EMstopSwitch(			TriggerInput := NOT (get.b_EstopChannelAOK AND get.b_EstopChannelBOK), 
						LogItemGroup :=  eLogItemGroupID.Safety, 
						LogItemName := 'EmStopSwCnt', 
						LogType := eLogTypes.TrackCycles);

SafetyStopCount(		TriggerInput := get.b_SafetyOK, 
						LogItemGroup :=  eLogItemGroupID.Safety, 
						LogItemName := 'SafetyStopCnt', 
						LogType := eLogTypes.TrackCycles);
END_METHOD

METHOD Reset : BOOL
VAR_INPUT
	prgReset: BOOL;
END_VAR
IF ton_Reset.Q THEN
	ToSafetyPrg.b_safetyPRGReset := FALSE;
	ToSafetyPrg.b_ErrorReset := FALSE;
	ton_Reset.IN := FALSE;
	Reset := get.b_SafetyOK;
ELSE
	ton_Reset.IN :=TRUE;
	ToSafetyPrg.b_safetyPRGReset := prgReset;
	ToSafetyPrg.b_ErrorReset := TRUE;
END_IF
END_METHOD

END_PROGRAM

// ---- POUs/Objects/WearLogging/FB_Varlogger.TcPOU
//FB for complex logvalues
//Can keep track of on-time, rising edge count, highest/lowest value and actual values
//Simple overwriting and min/max of variables can also be done without this by calling the Wearlogging methods directly

FUNCTION_BLOCK FB_Varlogger
VAR_INPUT
	LogItemGroup	:	eLogItemGroupID;		//Json itemgroup
	LogItemName		:	STRING;					//Json itemname
	LogType			:	eLogTypes;				//Determines logging functionality
	
	TriggerInput	:	BOOL;					//boolean input for trackcycles and trackOnTime
	NewValue		:	ANY;					//New value for 
END_VAR

VAR
	rtrig_InputValue		:	r_trig;
	ton_IncrementingTimer	:	ton	:=	(pt := T#15M);
	ftrig_timerloss			:	f_trig;
	rtrig_TimerDone			:	r_trig;
	elapsedTime				:	TIME;	
	
	ton_UpdateTimer			:	Ton;
	LrealPointer			: 	POINTER TO LREAL;
	realPointer				:	POINTER TO REAL;
	StringPointer			:	POINTER TO STRING;
	
	USINTPOINTER			: 	POINTER TO USINT;
	UINTPOINTER				: 	POINTER TO UINT;
	UDINTPOINTER			: 	POINTER TO UDINT;
	ULINTPOINTER			: 	POINTER TO ULINT;
	SINTPOINTER				: 	POINTER TO SINT;
	INTPOINTER				: 	POINTER TO INT;
	DINTPOINTER				: 	POINTER TO DINT;
	LINTPOINTER				: 	POINTER TO LINT;	

	TempString				:	String;	
END_VAR

CASE LogType OF 
	eLogTypes.TrackCycles:
		rtrig_InputValue(clk := TriggerInput);
		IF rtrig_InputValue.Q AND NOT gvl.b_Initcycle THEN
			WearLogging.SetInteger(LogItemGroup, LogItemName, LogType, 1);
		END_IF

	eLogTypes.TrackOnTime:
		ton_IncrementingTimer	(in := TriggerInput AND NOT ton_incrementingTimer.Q);
		ftrig_timerloss(clk := TriggerInput);
		rtrig_timerDone(clk := ton_IncrementingTimer.Q);
		
		IF ftrig_timerloss.Q THEN
			WearLogging.setFloat(LogItemGroup, LogItemName, LogType, TO_LREAL(TIME_TO_LREAL(elapsedTime)/TIME_TO_LREAL(T#1H)));
		END_IF
		
		IF rtrig_timerDone.Q THEN
			elapsedTime := ton_IncrementingTimer.PT;
			WearLogging.setFloat(LogItemGroup, LogItemName, LogType, TO_LREAL(TIME_TO_LREAL(elapsedTime)/TIME_TO_LREAL(T#1H)));
		END_IF
		
		elapsedTime := ton_IncrementingTimer.ET;
		
	eLogTypes.WriteValue, eLogTypes.KeepHighestValue, eLogTypes.KeepLowestValue:
		IF TriggerInput and not gvl.b_initCycle then	
		
			CASE NewValue.TypeClass OF
				__SYSTEM.TYPE_CLASS.TYPE_REAL:
					realPointer := NewValue.pValue;
					WearLogging.setFloat(LogItemGroup, LogItemName, LogType,TO_LREAL(realPointer^));
					
				__SYSTEM.TYPE_CLASS.TYPE_LREAL:
					LrealPointer := NewValue.pValue;
					WearLogging.setFloat(LogItemGroup, LogItemName, LogType,LrealPointer^);
					
				__SYSTEM.TYPE_CLASS.TYPE_USINT:
					USINTPOINTER := NewValue.pValue;
					WearLogging.setInteger(LogItemGroup, LogItemName, LogType, TO_LINT(USINTPOINTER^));
				
				__SYSTEM.TYPE_CLASS.TYPE_UINT:
					UINTPOINTER := NewValue.pValue;
					WearLogging.setInteger(LogItemGroup, LogItemName, LogType, TO_LINT(UINTPOINTER^));
				
				__SYSTEM.TYPE_CLASS.TYPE_UDINT:
					UDINTPOINTER := NewValue.pValue;
					WearLogging.setInteger(LogItemGroup, LogItemName, LogType, TO_LINT(UDINTPOINTER^));
				
				__SYSTEM.TYPE_CLASS.TYPE_ULINT:
					ULINTPOINTER := NewValue.pValue;
					WearLogging.setInteger(LogItemGroup, LogItemName, LogType, TO_LINT(ULINTPOINTER^));
				
				__SYSTEM.TYPE_CLASS.TYPE_SINT:
					SINTPOINTER := NewValue.pValue;
					WearLogging.setInteger(LogItemGroup, LogItemName, LogType, TO_LINT(SINTPOINTER^));
				
				__SYSTEM.TYPE_CLASS.TYPE_INT:
					INTPOINTER := NewValue.pValue;
					WearLogging.setInteger(LogItemGroup, LogItemName, LogType, TO_LINT(INTPOINTER^));
				
				__SYSTEM.TYPE_CLASS.TYPE_DINT:
					DINTPOINTER := NewValue.pValue;
					WearLogging.setInteger(LogItemGroup, LogItemName, LogType, TO_LINT(DINTPOINTER^));
				
				__SYSTEM.TYPE_CLASS.TYPE_LINT:
					LINTPOINTER := NewValue.pValue;
					WearLogging.setInteger(LogItemGroup, LogItemName, LogType, TO_LINT(LINTPOINTER^));

				__SYSTEM.TYPE_CLASS.TYPE_string:
					StringPointer := NewValue.pValue;
					TempString := StringPointer^;
					WearLogging.SetString(LogItemGroup, LogItemName, TempString);
			END_CASE
		END_IF
END_CASE

END_FUNCTION_BLOCK

// ---- POUs/Objects/WearLogging/WearLogging.TcPOU
PROGRAM WearLogging
VAR
	LoggerInitialized			:	Bool;
	ton_FileUpdateTime			:	Ton	:=	(pt := T#30M);
	WearLoggerState				:	LogState	:=	LogState.Init;
	fbJson						:	FB_JsonDynDomParser;
	FileName					:	STRING	:=	'C:\Users\Administrator\Documents\ePU10WearLogging.json';
	
	bLoad						:	BOOL;
	b_Saved						: 	BOOL;
	TON_FileTimer				:	Ton := (PT:= T#500MS);
	bLoaded						:	BOOL;
	JsonText					:	STRING(2000);
	JsonTextSize				: 	UDINT;
	SystemBootCountLogged		: 	BOOL := FALSE;

	Error						:	HResult;
	
	bexecWrite					:	BOOL;
	
	b_ForceWrite				:	Bool;
	b_Test						:	BOOL;
	JsonRoot					:	SJsonvalue;
	TempString					:	STring;
END_VAR


VAR
	SystemOnTime	:	FB_Varlogger;
	SystemOnCycles	:	FB_Varlogger;
	LogTimestamp	:	FB_Varlogger;
	TestLogger		:	FB_Varlogger;
END_VAR

VAR
	testString	:	STRING;
END_VAR

ton_FileUpdateTime();
ton_FileTimer();

CASE WearLoggerState OF
	LogState.Init:
		ton_FileTimer.in := NOT bLoad; //wait before initialising the logger
		IF ton_FileTimer.Q THEN
			bLoad := TRUE;
			bLoaded := FALSE;
			WearLoggerState := LogState.Loading_file;
		END_IF
				
	 LogState.Loading_file:	
	 	bLoaded := fbJson.LoadDocumentFromFile(FileName, bLoad, hrErrorCode=>Error);
		IF NOT bLoad THEN
			IF bLoaded THEN
				bLoaded := FALSE;
				LocalItems();
				JsonTextSize := fbJson.CopyDocument(JsonText, SIZEOF(JsonText));
				WearLoggerState := Logstate.Idle;
			ELSIF Error = 16#9811070C OR Error = 16#00000001 THEN
				WearLoggerSTate := Logstate.FileNotFound;
			END_IF
		END_IF
			
	LogState.Idle:
		fbJson.SetMaxDecimalPlaces(3);
		ton_FileUpdateTime.IN := TRUE;
		IF ton_FileUpdateTime.Q OR b_ForceWrite THEN
			JsonTextSize := fbJson.CopyDocument(JsonText, SIZEOF(JsonText));
			WearLoggerState := LogState.SavingLogData;
			bexecWrite := TRUE;
		END_IF
		
	Logstate.SavingLogData:	
		b_Saved := fbJson.SaveDocumentToFile(FileName, bexecWrite, hrErrorCode=>Error);
		IF NOT bexecWrite THEN
			IF b_Saved THEN
				b_ForceWrite :=	FALSE;
				ton_FileUpdateTime.IN := FALSE;
			END_IF
			WearLoggerState := LogState.Idle;
		END_IF
		
	LogState.FileNotFound: //File not found, create empty JSON and try again.
		fbJson.NewDocument();
		JsonRoot := fbjson.GetDocumentRoot();
		tempString := concat(gvl.s_SystemDate, ' ');
		tempString := concat(tempSTring, gvl.s_SystemTime);
		SetString(eLogItemGroupID.General, 'LogCreationDate', tempString);
	
		bexecWrite := TRUE;
		b_Saved := fbJson.SaveDocumentToFile(FileName, bexecWrite, hrErrorCode=>Error);
		IF NOT bexecWrite THEN
				WearLoggerState := LogState.Init;
		END_IF		
END_CASE


IF WearLoggerstate = Logstate.SavingLogData OR WearLoggerstate = Logstate.Idle THEN
	main_fast.ACswitchgear.GetWearCounters();
	main_fast.Coolingsystem.GetWearCounters();
	main_fast.BMS.GetWearCounters();
	main_fast.PowerStack.GetWearCounters();
	main_fast.Enclosure.GetWearCounters();
	main_fast.InternalPowerSupply.GetWearCounters();
	safety.GetWearCounters();
	LocalItems();
END_IF

METHOD PRIVATE CreateLogEntry : sJsonValue
VAR_INPUT
	e_LogItemGroup		:	eLogItemGroupID;
	s_LogItemName		:	STRING;
	EntryType			:	eEntryType;
END_VAR

VAR
	s_LogItemGroup		:	STRING;
	JsonPath			:	STRING;
	LogEntry			:	sJsonValue;
	JsonRoot			:	sjsonValue;
END_VAR

VAR_OUTPUT
	//LogEntry	:	sJsonValue;
END_VAR
JsonRoot := fbjson.GetDocumentRoot();
LogEntry := JsonRoot;

//empty LogItemGroup not allowed, group.none removed.
s_LogItemGroup := TO_STRING(e_LogItemGroup);
LogEntry := fbJson.FindMember(JsonRoot, s_LogItemGroup);
IF LogEntry = 0 THEN //member doesn't exist, create empty Json;
	LogEntry := fbJson.AddJsonMember(JsonRoot, s_LogItemGroup, '');
ELSE
	IF NOT fbJson.isObject(LogEntry) THEN
		LogEntry := fbJson.AddJsonMember(JsonRoot, s_LogItemGroup, '');
	END_IF
END_IF


CASE EntryType OF
	eEntryType.IntegerValue:
		CreateLogEntry := fbJson.AddInt64Member(LogEntry, s_LogItemName, 0);
	eEntryType.FloatValue:
		CreateLogEntry := fbJson.AddDoubleMember(LogEntry, s_LogItemName, 0.000);
	eEntryType.StringValue:
		CreateLogEntry := fbJson.AddStringMember(LogEntry, s_LogItemName, '1970-01-01 00:00:00.000');
END_CASE
END_METHOD

METHOD GetFloatValue : BOOL
VAR_INPUT
	e_LogItemGroup		:	eLogItemGroupID;
	s_LogItemName		:	STRING;
END_VAR

VAR_OUTPUT
	CurrentLogValue		:	LREAL;
END_VAR

VAR
	jsonItem		:	SJsonValue;
	JSonString		:	STRING(2000);
	CurrentValue 	: 	LREAL 		:= 0;
	IsNewValue		:	Bool;
END_VAR
//Maybe add a check if the new value is higher than the old one;
IF getLogEntry(e_LogItemGroup, s_LogItemName, eEntryType.FloatValue, LogEntry => jsonItem, IsNewValue => IsNewValue) THEN
	CurrentLogValue := fbJson.GetDouble(JsonItem);
END_IF
END_METHOD

METHOD GetLogEntry : BOOL
VAR_INPUT
	e_LogItemGroup		:	eLogItemGroupID;
	s_LogItemName		:	STRING;
	EntryType			:	eEntryType;
END_VAR

VAR
	s_LogItemGroup	:	STRING;
	JsonPath		:	STRING;
	JsonRoot		:	sjsonValue;
END_VAR

VAR_OUTPUT
	LogEntry	:	SJsonValue;
	IsNewValue	:	Bool;
END_VAR
GetLogEntry	:=	FALSE;
jsonRoot := fbJson.GetDocumentRoot();

//empty path not allowed due to difficulties with OR integration.
//So always get LogItemGroup first
JsonPath := concat(TO_STRING(e_LogItemGroup), '/');
JsonPath := concat(JsonPath, TO_STRING(s_LogItemName));
LogEntry := fbJson.FindMemberPath(jsonRoot, JsonPath);	
LogEntry;


IF (LogEntry = 0) THEN
	LogEntry := CreateLogEntry(e_LogItemGroup, s_LogItemName, EntryType);
	IsNewValue := TRUE;
	GetLogEntry := TRUE; 
	Logentry;
ELSE
	CASE EntryType OF
		eEntryType.IntegerValue:
			IF  fbJson.IsInt64(LogEntry) THEN
				GetLogEntry := TRUE; 
			END_IF //return fail if wrong variable type already exists with this name. Not sure what to do now.
		eEntryType.FloatValue:
			IF  fbJson.IsDouble(LogEntry) THEN
				GetLogEntry := TRUE; 
			END_IF //return fail if wrong variable type already exists with this name. Not sure what to do now.
		eEntryType.StringValue:
			//IF  fbJson.IsString(LogEntry) THEN
				GetLogEntry := TRUE; 
			//END_IF //return fail if wrong variable type already exists with this name. Not sure what to do now.	
	END_CASE
END_IF
END_METHOD

METHOD LocalItems : BOOL
VAR_INPUT
END_VAR
SystemOnTime(		TriggerInput := TRUE, 
					LogItemGroup :=  eLogItemGroupID.General, 
					LogItemName := 'SystemOnTime', 
					LogType := eLogTypes.TrackOnTime);

SystemOnCycles(		TriggerInput := NOT SystemBootCountLogged, 
					LogItemGroup :=  eLogItemGroupID.General, 
					LogItemName := 'SystemCycles', 
					LogType := eLogTypes.TrackCycles);

tempString:= concat(gvl.s_SystemDate, concat(' ', gvl.s_SystemTime));
SetString(eLogItemGroupID.General, 'LogTimestamp', tempString);

SetString(eLogItemGroupID.General, 'PlcSwVer', settings.Properties.s_SWversionNumber);

TestLogger(			TriggerInput := b_Test, 
					LogItemGroup :=  eLogItemGroupID.General, 
					LogItemName := 'StringTest', 
					LogType := eLogTypes.WriteValue,
					NewValue := testString);

b_test := FALSE;

SystemBootCountLogged := TRUE;
END_METHOD

METHOD SetFloat : BOOL
VAR_INPUT
	e_LogItemGroup		:	eLogItemGroupID;
	s_LogItemName		:	STRING;
	LogType				:	eLogTypes;
	Value				:	LREAL;
END_VAR

VAR
	jsonItem		:	SJsonValue;
	JSonString		:	STRING(2000);
	CurrentValue 	: 	LREAL 		:= 0;
	IsNewValue		:	Bool;
END_VAR
//Maybe add a check if the new value is higher than the old one;
IF getLogEntry(e_LogItemGroup, s_LogItemName, eEntryType.FloatValue, LogEntry => jsonItem, IsNewValue => IsNewValue) THEN
	
	CurrentValue := fbJson.GetDouble(JsonItem);
	
	CASE LogType OF
		eLogTypes.TrackOnTime:
			jsonItem := fbJson.SetDouble(jsonItem, CurrentValue+Value);
			
		eLogTypes.KeepHighestValue:
			IF (Value > CurrentValue) OR IsNewValue THEN
				jsonItem := fbJson.SetDouble(jsonItem, Value);
			END_IF
			
		eLogTypes.KeepLowestValue:
			IF (Value < CurrentValue) OR IsNewValue THEN
				jsonItem := fbJson.SetDouble(jsonItem, Value);
			END_IF
			
		eLogTypes.WriteValue:
			jsonItem := fbJson.SetDouble(jsonItem, Value);
	END_CASE
END_IF
END_METHOD


METHOD SetInteger : BOOL
VAR_INPUT
	e_LogItemGroup		:	eLogItemGroupID;
	s_LogItemName		:	STRING;
	LogType				:	eLogTypes;
	Value				:	LINT;
END_VAR

VAR
	jsonItem		:	SJsonValue;
	JSonString		:	STRING(2000);
	CurrentValue 	: 	LINT 		:= 0;
	IsNewValue		:	Bool;
END_VAR
//Maybe add a check if the new value is higher than the old one;
IF getLogEntry(e_LogItemGroup, s_LogItemName, eEntryType.IntegerValue, LogEntry => jsonItem, IsNewValue => IsNewValue) THEN
	
	CurrentValue := fbJson.Getint64(JsonItem);
		
	CASE LogType OF
		eLogTypes.TrackCycles:
			jsonItem := fbJson.Setint64(jsonItem, CurrentValue+1);
			
		eLogTypes.KeepHighestValue:
			IF (Value > CurrentValue) OR IsNewValue THEN
				jsonItem := fbJson.Setint64(jsonItem, Value);
			END_IF
			
		eLogTypes.KeepLowestValue:
			IF (Value < CurrentValue) OR IsNewValue THEN
				jsonItem := fbJson.Setint64(jsonItem, Value);
			END_IF
			
		eLogTypes.WriteValue:
			jsonItem := fbJson.Setint64(jsonItem, Value);
	END_CASE
END_IF
END_METHOD

METHOD SetString : BOOL
VAR_INPUT
	e_LogItemGroup		:	eLogItemGroupID;
	s_LogItemName		:	STRING;
END_VAR

VAR_IN_OUT CONSTANT
	LogValue			:	STRING;
END_VAR

VAR
	jsonItem		:	SJsonValue;
END_VAR
//setDatetime doesn't seem to work. Changed to string for now
IF getLogEntry(e_LogItemGroup, s_LogItemName, eEntryType.StringValue, LogEntry => jsonItem) THEN
	JsonItem := fbJson.SetString(JsonItem, LogValue);
END_IF
END_METHOD

METHOD SystemShutdown : BOOL
VAR_INPUT
END_VAR
b_forceWrite := TRUE;
END_METHOD

END_PROGRAM

// ---- POUs/MonitoringControl/ControlManager.TcPOU
PROGRAM ControlManager
VAR_OUTPUT PERSISTENT
	PLCpersistvars				: ST_PLCPersistentvars;
END_VAR

VAR_IN_OUT
	control						: ST_ControlVars;
	Operation					: ST_OperationVars;
END_VAR

VAR
	{ attribute 'TcHmiSymbol.Show' }
	IoT							: FB_IotController;	
	PNController				: FB_ExternalController;
	TestScripts					: FB_Testscripts;	
END_VAR

VAR_IN_OUT CONSTANT
	{ attribute 'TcHmiSymbol.Hide' }
	monitor						: ST_System_Monitor;
END_VAR

//For persistentvars method
VAR
	
	fb_WritePersistentData		: WritePersistentData;
	r_trigWritePersistent		: R_TRIG;
	f_trigPersistentSucces		: F_Trig;
	b_PersistentWritten			: BOOL;
END_VAR

//instantiate fbs
//Call HMI program 
hmi(monitor:=monitor,
	PNControlvars := PnController.get,
	IotControlvars:= Iot.get,
	PLCpersistvars	:= PLCpersistvars);

//Call PNcontroller FB
PNController(monitor := monitor, st_params := Settings.MachineParams.PNController,
	controlvars := HMI.Controlvars);
	PNcontroller.set.b_available := settings.Configuration.e_PNcouplerType <> ePNcouplerType.None;
	
//Call IoT FB
Iot(monitor:=monitor, st_params:= settings.MachineParams.IOT,
	controlvars := HMI.Controlvars, a_ActiveEvents := Errorhandling.a_ActiveEvents);

//Test scripts	
TestScripts(monitor := monitor, controlvars := HMI.Controlvars);

//Select  Control source
ControlSourceSelector();



//WRITE PERSISTENT DATA
r_trigWritePersistent(CLK:= HMI.Controlvars.control.b_ActivateSettings);
f_trigPersistentSucces(CLK := fb_WritePersistentData.BUSY);
fb_WritePersistentData(NETID := '', PORT:= 851, START:=r_trigWritePersistent.Q,  TMOUT := T#5S);

IF f_trigPersistentSucces.Q AND NOT fb_WritePersistentData.ERR THEN
	b_PersistentWritten := TRUE;
ELSIF r_trigWritePersistent.Q THEN
	b_PersistentWritten := FALSE;
END_IF

METHOD PROTECTED ControlSourceSelector
IF HMI.controlvars.control.b_ActivateSettings or hmi.Controlvars.HMIonly.b_ActivateSetting THEN
	IF monitor.b_modeSwitchEnable THEN
		PLCpersistvars.Hardsettings := HMI.controlvars.HardSettings;
	END_IF
END_IF

//Fixed binding
control		:= HMI.Controlvars.control;
Operation	:= HMI.controlvars.Operation;


IF (MEMCMP(ADR(HMI.controlvars.Softsettings), ADR(PLCpersistvars.Softsettings), SIZEOF(PLCpersistvars.Softsettings)) <> 0) THEN
	PLCpersistvars.Softsettings	:= HMI.controlvars.SoftSettings;
END_IF
END_METHOD

END_PROGRAM

// ---- POUs/MonitoringControl/IoT/FB_IotController.TcPOU
FUNCTION_BLOCK FB_IotController
VAR_OUTPUT
	get								: ST_ExtController_get;
END_VAR

VAR_IN_OUT CONSTANT
	{ attribute 'TcHmiSymbol.Hide' }
	monitor								: ST_System_Monitor;
END_VAR

//HMI controls to be overwritten from get if controller is allowed.
VAR_IN_OUT
	controlvars							: ST_System_Control;
	st_params							: ST_IOT_params;
	a_activeEvents						: ARRAY [*] OF ST_errorstruct;
END_VAR


VAR
	BindControlVars						: FB_BindControlvars;
	ListUpdated							: BOOL;
	FBAssetConfig						: RestComOpenremote;
END_VAR

VAR PERSISTENT
	{ attribute 'TcHmiSymbol.ShowRecursively' }
	IotDataSharingList					: ARRAY [1..2000] OF ST_IoTDataHMI;
	{ attribute 'TcHmiSymbol.ShowRecursively' }
	CreditCoverage						: ST_IotData_credits;
END_VAR

VAR
	FBJSON	 : FB_JsonDomParser;
	bWriteToFile	:	BOOL;
	bresult	:	BOOL;
	error : HRESULT;
	length : UDINT;
	output	:	STRING(10000);
	filename	:STRING :='C:\PLCUtility\IoTDataSharing.json';
END_VAR

// Fill IotDatasharing array
IF CreateIoTDataList(SaveJson := controlvars.control.b_ActivateIotSettings, aData:= IotDataSharingList) THEN
	Listupdated:= TRUE;
	controlvars.control.b_ActivateIotSettings := FALSE;
END_IF

//Provisioning
FBAssetConfig(monitor:= monitor, controlvars:= get, st_params:= st_params, HMILogData := IotDataSharingList, UpdateConfiguration := Listupdated, IOTCredits := CreditCoverage);

IF FBAssetConfig.ConfigurationDone THEN
	get.LoggingBudgetOK := (CreditCoverage.RemainingCredits >= 0);
		
	// CALL MQTT PROGRAM
	MqttComOpenremote(updatetrigger:= listupdated, monitor:= monitor, controlvars:= get, st_params:= st_params, aData:= IotDataSharingList);
	Listupdated := FALSE;
	//Build message for MQTT
	MessageBuilder(SIZEOF(MqttComOpenremote.sEventMsg), ADR(MqttComOpenremote.sEventMsg), a_activeEvents, MqttComOpenRemote.eActiveMsg);
	
	//BIND CONTROLVARS TO HMI CONTROL VARS IF IOT CONTROL IS ENABLED BY USER
	IF st_params.b_controlEnable AND monitor.controlfb.HardSettings.setup.e_ControlSource = eControlsources.PowerNet THEN
		BindControlvars(
				advancedcontrol := get.b_AdvancedControl, 
				Systemcontrolvars := controlvars,
				ExtControlvars := get);
	END_IF
	
	//GET FEEDBACK OF STATE.3
	get.b_Active := MqttComOpenremote.fbMqttClient.bConnected;
	get.e_ConnectionState := mqttComOpenRemote.e_state;
END_IF

METHOD CreateIoTDataList : BOOL
VAR_INPUT
	saveJson	: BOOL;
END_VAR

VAR_INST
	init :BOOL := TRUE;
	initJson :BOOL := TRUE;
	executeJson : BOOL;
END_VAR
VAR_IN_OUT
	aData			: ARRAY [*] OF ST_IotDataHMI;
END_VAR

VAR
	index			: DINT;
END_VAR

VAR_INST
	b_loaded : BOOL;
END_VAR

CreateIoTDataList := FALSE;
IF init THEN
	// Set varnames in array slots
	FOR index := (eDataMappingVarNames.none +1) TO MIN(UPPER_BOUND(aData,1), eDataMappingVarNames.last -1) DO
		aData[index].Varname := index;
		IF FIND(TO_STRING(aData[index].varname), 'controlfb') = 1 THEN
			aData[index].b_IOTWriteAllowed := TRUE;
		END_IF	
	END_FOR;
	init := FALSE;
	initJson := TRUE;
END_IF




CreateIoTDataList := DiskToFromJsonFile(
		PathName 	:= filename,
		read 			:= initJson OR settings.Load, 
		write 			:= SaveJson, 
		aData 			:= aData
) OR SaveJson;
//CreateIoTDataList :=  SaveJson;

IF CreateIoTDataList THEN
	initJson := FALSE;
END_IF
END_METHOD

METHOD DiskToFromJsonFile : BOOL
VAR_INPUT
	Pathname	: STRING := 'C:\PLCUtility\IoTDataSharing.json';
	write			: BOOL;
	read			: BOOL;
END_VAR

VAR_IN_OUT
	aData			: ARRAY [*] OF ST_IotDataHMI;
END_VAR

VAR_INST
	sJsonPathname	: STRING := 'C:\PLCUtility\IoTDataSharing.json';
    // Triggers
    TrigReadFromDisk  : R_TRIG;
    TrigWriteToDisk   : R_TRIG;

    // Status / result
    b_Error           : BOOL;
    Error             : HRESULT;
    Counter           : UINT;

    // Async control
    WriteToDisk       : BOOL;
    ReadFromDisk      : BOOL;

    // State machine
    State             : UINT;   // 0=idle, 10=prepare save, 20=save busy, 30=load busy, 40=parse loaded json, 900=error
    MaxIndex          : DINT;

    // JSON handling
    version           : STRING(4) := '1.0';
   // fbJson            : FB_JsonDomParser;
    jsonDoc           : SJsonValue;
    jsonRoot          : SJsonValue;
    jsonItem          : SJsonValue;
	jsonSubItem		  : SJsonValue;

    // Temp vars
    tempString        : STRING(255);
	structname			: STRING := 'ST_IotDataHMI';
    sJson             : STRING(2000);
    index             : DINT;
    bOk               : BOOL;
	
	length	:	UDINT;

	b_Saved           : BOOL;
    b_Loaded          : BOOL;
END_VAR
// -----------------------------------------------------------------------------
// Edge detection
// -----------------------------------------------------------------------------
TrigReadFromDisk(CLK := read);
TrigWriteToDisk(CLK := write);

IF TrigReadFromDisk.q THEN
	b_loaded := FALSE;
	//sJsonPathName := Pathname;
END_IF

IF TrigWriteToDisk.Q THEN
	b_saved := FALSE;
	//sJsonPathName := Pathname;
END_IF

// -----------------------------------------------------------------------------
// Default return
// -----------------------------------------------------------------------------
//DiskToFromJsonFile := FALSE;

// -----------------------------------------------------------------------------
// State machine
// -----------------------------------------------------------------------------
CASE State OF

    // -------------------------------------------------------------------------
    // IDLE
    // -------------------------------------------------------------------------
    0:
        // Clear one-shot result flags only when idle
        b_Error := FALSE;
        Error := 0;
        Counter := 0;

        // Compute upper loop bound once
        MaxIndex := UPPER_BOUND(aData, 1);
        IF MaxIndex > (TO_DINT(eDataMappingVarNames.last) - 1) THEN
            MaxIndex := TO_DINT(eDataMappingVarNames.last) - 1;
        END_IF;
		
       IF read AND NOT b_loaded THEN
		   ReadFromDisk := TRUE;
           State := 30;
	   ELSIF write AND NOT b_saved THEN
		   State := 10;
	   END_IF
	  


    // -------------------------------------------------------------------------
    // PREPARE SAVE DOCUMENT
    // -------------------------------------------------------------------------
    10:
        fbJson.NewDocument();
        jsonRoot := fbJson.GetDocumentRoot();

        // Root must be an object before adding members
       //JsonObject = fbJson.SetObject(jsonRoot);

        tempString := CONCAT(gvl.s_SystemDate, ' ');
        tempString := CONCAT(tempString, gvl.s_SystemTime);

        fbJson.AddStringMember(jsonRoot, 'creationDate', tempString);
        fbJson.AddStringMember(jsonRoot, 'version', version);

        FOR index := TO_DINT(eDataMappingVarNames.none) + 1 TO MaxIndex DO
            IF aData[index].Varname <> 0 THEN
                tempString := TO_STRING(aData[index].Varname);
                jsonItem := fbJson.AddObjectMember(jsonRoot, tempString);
				fbJson.AddStringMember(jsonItem, 'Label', aData[index].Label);
                fbJson.AddUintMember(jsonItem, 'LogType', aData[index].LogType);
                fbJson.AddUintMember(jsonItem, 'LogInterval', aData[index].LogInterval);
				fbJson.AddStringMember(jsonItem, 'Unit', aData[index].Unit); 
            END_IF
        END_FOR

        //WriteToDisk := TRUE;
		bWriteToFile := TRUE;
        State := 20;


    // -------------------------------------------------------------------------
    // SAVE BUSY
    // Keep WriteToDisk TRUE until operation finishes or errors
    // -------------------------------------------------------------------------
    20:

		//IF bWriteToFile THEN
			bresult := fbJson.SaveDocumentToFile(
				sFile      := sJsonPathname,
				bExec      := bWriteToFile,
				hrErrorCode => Error
			);
		IF NOT bWriteToFile THEN//WriteToDisk THEN
			IF Error = 0 THEN
				b_Saved := TRUE;
				//DiskToFromJsonFile := TRUE;
				State := 0;
			ELSE
				b_Error := TRUE;
				State := 900;
			END_IF
        END_IF


    // -------------------------------------------------------------------------
    // LOAD BUSY
    // Keep ReadFromDisk TRUE until operation finishes or errors
    // -------------------------------------------------------------------------
    30:
        bOk := fbJson.LoadDocumentFromFile(
            sFile      := sJsonPathname,
            bExec      := ReadFromDisk,
            hrErrorCode => Error
        );

        IF NOT ReadFromDisk THEN
            IF Error = 0 THEN
            	State := 40;
			ELSE
				// Optional: if file missing / invalid, regenerate from current data
				// Keep this only if you really want auto-create behavior
				IF (Error = -1743714548 ) OR (Error = 16#00000001) THEN //16#9811070C
					Error := 0;
					State := 10; // create and save a fresh file
				ELSE
					b_Error := TRUE;
					State := 900;
				END_IF
			END_IF
        END_IF


    // -------------------------------------------------------------------------
    // PARSE LOADED JSON INTO ARRAY
    // -------------------------------------------------------------------------
    40:
        jsonRoot := fbJson.GetDocumentRoot();
        Counter := 0;
        //b_Loaded := FALSE;

        FOR index := TO_DINT(eDataMappingVarNames.none) + 1 TO MaxIndex DO
            IF aData[index].Varname <> 0 THEN
                tempString := TO_STRING(aData[index].Varname);
                jsonItem := fbJson.findMember(jsonRoot, tempString);

                IF jsonItem <> 0 THEN
					 // LogType
					jsonSubItem := fbJson.FindMember(jsonItem, 'LogType');
					IF jsonSubItem <> 0 THEN
						aData[index].LogType := TO_UINT(fbJson.GetUint(jsonSubItem));
					END_IF
	
					// LogInterval
					jsonSubItem := fbJson.FindMember(jsonItem, 'LogInterval');
					IF jsonSubItem <> 0 THEN
						aData[index].LogInterval := TO_UINT(fbJson.GetUint(jsonSubItem));
					END_IF
	
					// Unit
					jsonSubItem := fbJson.FindMember(jsonItem, 'Unit');
					IF jsonSubItem <> 0 THEN
						aData[index].Unit := fbJson.GetString(jsonSubItem);
					END_IF
	
					// Label
					jsonSubItem := fbJson.FindMember(jsonItem, 'Label');
					IF jsonSubItem <> 0 THEN
						aData[index].Label := fbJson.GetString(jsonSubItem);
					END_IF
	
					Counter := Counter + 1;
                END_IF
            END_IF
        END_FOR

        // Consider load successful if at least one item was restored
        IF Counter > 0 THEN
            b_Loaded := TRUE;
            DiskToFromJsonFile := TRUE;
            State := 0;
        ELSE
            // If file loaded but no matching members found, recreate it
            State := 10;
        END_IF


    // -------------------------------------------------------------------------
    // ERROR
    // -------------------------------------------------------------------------
    900:
        b_Error := TRUE;
       // DiskToFromJsonFile := TRUE;
       // State := 0;

END_CASE;
END_METHOD

METHOD FindJsonMember : BOOL
VAR_INPUT
END_VAR
END_METHOD

METHOD GetDiagnostics 
VAR_IN_OUT
	AddError		: ARRAY [*] OF FB_AddErrorST;
	a_ActiveEvents	: ARRAY [*] OF ST_ErrorStruct;
	w_Index			: WORD;
END_VAR
(*IPS*)
	(*AC PSU fault*)		AddError[w_Index](
			b_ErrorTrig			:= NOT get.LoggingBudgetOK,
			out_ST_Error		:= a_ActiveEvents[w_Index],
			w_ErrorID			:= 1,
			e_objectID			:= eObject_ID.IotController,
			s_Message			:= 'Logging budget exceeded. Logging halted until configuration is valid',
			e_sev				:= eSeverity.Warning,
			t_triggerTime		:= T#1S,
			b_AutoClear			:= TRUE
			);
		//w_Index := w_Index +1;
END_METHOD

METHOD MessageBuilder

VAR_INPUT
	nSize								: UDINT;
	sMsg 								: POINTER TO STRING;
END_VAR

VAR_IN_OUT
	a_activeEvents						: ARRAY [*] OF ST_errorstruct;
	eActiveMsg							: eSeverity; // range from 0 to 5. 0 = none, 1 info, ... 5 em shutdown
END_VAR

VAR_INST
	i_RequiredLength			: INT; //Messages from Emergency Shutdown, Quick Shutdown and Normal Shutdown.
	w_MessageCheckSum			: WORD;
	w_MessageCheckSumLast		: WORD;
	bMsgFull					: BOOL;
	di_nElements				: DINT;
	bOnChange					: BOOL;
	//sMsg						: STRING(1000);
	s_EndMessage				: STRING(13):= ', and more...';
	s_messageBreak				: STRING(3) := '\n'; 
	s_messageSeparation			: STRING(3) := ',  '; 
	b_ClearMessage				: BOOL;
	
	by_currentIndex				: BYTE;
	a_ErrorIndex				: ARRAY[0..10] OF WORD;
	by_SortedIndex				: BYTE;
	a_ErrorIndexSorted			: ARRAY[0..10] OF WORD;
END_VAR



VAR
	s_ErrorMessage	: STRING(256);
	s_sevtemp		: STRING(256) ;
	i 				: DINT;
	j 				: INT;
	s_filterName	: STRING;
	w_ErrorIndex	: WORD;
END_VAR
di_nElements := TO_DINT(nSize);// / SIZEOF(STRING(1));
by_currentIndex := 0; 
w_MessageCheckSum := 0; 


IF b_ClearMessage THEN
	sMsg^ := '';
END_IF

MEMSET(ADR(a_ErrorIndex), 0, SIZEOF(a_ErrorIndex));

//FIRST CHECK SOMETHING HAS CHANGED AND SAVE THE CORRESPONDING INDEXES SORTED BY SEVERITY
FOR i:= 0 TO UPPER_BOUND(a_ActiveEvents,1) DO
	IF a_ActiveEvents[i].b_ErrorActive AND a_ActiveEvents[i].s_Severity <> TO_STRING(eSeverity.Info) THEN
		//max 10 messages will be evaluated
		w_MessageCheckSum := w_MessageCheckSum + TO_WORD(i);
		IF by_currentIndex < 10 THEN
			a_ErrorIndex[by_CurrentIndex] := TO_WORD(i);
			by_currentIndex := by_currentIndex + 1;
		END_IF
	END_IF
END_FOR

bOnChange := w_MessageCheckSum <> w_MessageCheckSumLast;
w_MessageCheckSumLast := w_MessageCheckSum;

//IF CHANGED, SET STRINGS
IF bOnChange THEN
	//SORT on severity
	MEMSET(ADR(a_ErrorIndexSorted), 0, SIZEOF(a_ErrorIndexSorted));
	by_SortedIndex := 0; 
	FOR j:= 1 TO 4 DO
		//select filter
		CASE j OF
			1 : s_filterName := TO_STRING(eSeverity.EmergencyShutdown);
			2 : s_filterName := TO_STRING(eSeverity.QuickShutdown);
			3 : s_filterName := TO_STRING(eSeverity.NormalShutdown);
			4 : s_filterName := TO_STRING(eSeverity.Warning);
			5 : s_filterName := TO_STRING(eSeverity.Info);
		END_CASE
	
		FOR i:= 0 TO by_currentIndex -1 DO
			w_ErrorIndex := a_ErrorIndex[i];
			IF a_ActiveEvents[w_ErrorIndex].s_Severity = s_filtername THEN
				IF eactiveMsg < j THEN
					eActiveMsg := TO_BYTE(j);
				END_IF
				a_ErrorIndexSorted[by_SortedIndex] := a_ErrorIndex[i];
				by_SortedIndex := by_SortedIndex + 1;
			END_IF
		END_FOR
	END_FOR	
	
	//-------Message Formatter----------------------------------------------------------------------
	
	bMsgFull := FALSE;
	sMsg^ := '';
	s_SevTemp := '';
	FOR i:= 0 TO by_SortedIndex -1 DO
		w_ErrorIndex := a_ErrorIndexSorted[i];
	//clear message
		s_ErrorMessage := '';
	// Write Message
		IF s_sevtemp <> a_ActiveEvents[w_ErrorIndex].s_Severity THEN 
			s_ErrorMessage 	:= concat(s_ErrorMessage, a_ActiveEvents[w_ErrorIndex].s_Severity);
			s_ErrorMessage	:= concat(s_ErrorMessage, ': ');
			s_ErrorMessage	:= concat(s_ErrorMessage, s_messageBreak);
			s_sevtemp := a_ActiveEvents[w_ErrorIndex].s_Severity;
		END_IF
		s_ErrorMessage	:= concat(s_ErrorMessage, a_ActiveEvents[w_ErrorIndex].s_Message);
		i_RequiredLength := TO_INT(len2(pSTRING := sMsg)) + LEN(s_ErrorMessage);
		
		IF (i_RequiredLength < di_nElements - LEN(s_EndMessage)- LEN(s_endMessage)) THEN
			// Add comma and space if not first msg
			IF sMsg^ <> '' THEN
				concat2(pSrcString1 := sMsg,pSrcString2:=ADR(s_messageSeparation), pDstString := sMsg, nDstSize :=nSize);
			END_IF 
			//Add msg
			concat2(pSrcString1 := sMsg,pSrcString2:=ADR(s_ErrorMessage), pDstString := sMsg, nDstSize := nSize);
		ELSE
			//Trigger message is full
			IF NOT bMsgFull THEN
				concat2(pSrcString1 := sMsg,pSrcString2:=ADR(s_EndMessage), pDstString := sMsg, nDstSize := nSize);
			END_IF
			bMsgFull := TRUE;
			EXIT;
		END_IF
	END_FOR
END_IF

IF sMsg^ = '' AND w_MessageCheckSum <> 0 THEN
	w_MessageCheckSumLast := 0;
END_IF
END_METHOD

METHOD PresetBasicControl
VAR_INPUT
	enable				: BOOL;
END_VAR

VAR_INST
	rtrig_SetPreset		: r_Trig;
END_VAR


VAR_IN_OUT
	SoftOut		: ST_Softsettings;
END_VAR
rtrig_SetPreset(CLK:= enable);

IF rTrig_SetPreset.Q THEN
	SoftOut.system.b_EnableTransportMode := FALSE;
END_IF

SoftOut.system.b_AutomaticSwitching := TRUE;
END_METHOD

END_FUNCTION_BLOCK

// ---- POUs/Functions-FBs-Programs/Fb_BindControlVars.TcPOU
FUNCTION_BLOCK Fb_BindControlVars
VAR_INPUT
	AdvancedControl : BOOL;
END_VAR

VAR_IN_OUT
	SystemControlVars : ST_System_Control;
	ExtControlVars		: ST_ExtController_get;
END_VAR

VAR
	defaults			: ST_Softsettings;
	ftrig_AdvancedControl : F_trig;
	rTrig_AdvancedControl : R_Trig;
	
	b_defaultsRestored	: BOOL;
END_VAR

VAR
	WoE_Start		:	WriteOnEdge;
	WoE_Stop		:	WriteOnEdge;
	WoE_Activate	:	WriteOnEdge;
	WoE_Shutdown	:	WriteOnEdge;
	WoE_ClearHistory	:	WriteOnEdge;
	WoE_EMstop		:	WriteOnEdge;
	WoE_DehumStart	:	WriteOnEdge;
	WoE_Reset		:	WriteOnEdge;
END_VAR
VAR // added by the converter: edge detectors and wires of the graphical bodies
    _rt1, _rt2, _rt3, _rt4, _rt5, _rt6, _rt7, _rt8 : R_TRIG;
END_VAR

ftrig_AdvancedControl(CLK:= advancedcontrol);
IF ftrig_advancedControl.Q THEN
	RestoreDefaults(defaults, Systemcontrolvars.SoftSettings);
END_IF

//advanced control, all IO coupled
IF advancedcontrol THEN
	SystemControlVars.SoftSettings := ExtControlVars.SoftSettings;
	SystemControlVars.Operation := ExtControlVars.Operation;
ELSE
	Storedefaults(defaults, Systemcontrolvars.SoftSettings);
	//Basic control, only specific IO coupled
	Systemcontrolvars.softsettings.system.b_EcoModeEnable := ExtControlVars.SoftSettings.system.b_EcoModeEnable;
	SystemControlvars.operation.system.b_PFsetEnable := ExtControlVars.Operation.system.b_PFsetEnable;
	SystemControlvars.operation.system.r_PFset := ExtControlVars.Operation.system.r_PFset;
	SystemControlvars.operation.system.r_Pset:= ExtControlVars.Operation.system.r_Pset;
	SystemControlvars.operation.system.r_Qset:= ExtControlVars.Operation.system.r_Qset;
	SystemControlvars.softsettings.PSB.setpointTimeslot1 := ExtControlVars.softsettings.PSB.setpointTimeslot1;
END_IF

a_ControlCommands();

ACTION a_ControlCommands:
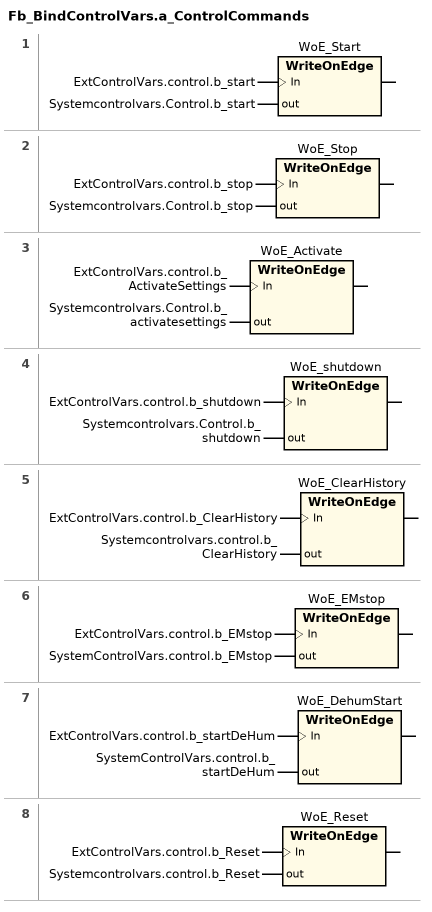
// NETWORK 1
_rt1(CLK := ExtControlVars.control.b_start);
WoE_Start(In := _rt1.Q, out := Systemcontrolvars.Control.b_start); // WriteOnEdge

// NETWORK 2
_rt2(CLK := ExtControlVars.control.b_stop);
WoE_Stop(In := _rt2.Q, out := Systemcontrolvars.Control.b_stop); // WriteOnEdge

// NETWORK 3
_rt3(CLK := ExtControlVars.control.b_ActivateSettings);
WoE_Activate(In := _rt3.Q, out := Systemcontrolvars.Control.b_activatesettings); // WriteOnEdge

// NETWORK 4
_rt4(CLK := ExtControlVars.control.b_shutdown);
WoE_shutdown(In := _rt4.Q, out := Systemcontrolvars.Control.b_shutdown); // WriteOnEdge

// NETWORK 5
_rt5(CLK := ExtControlVars.control.b_ClearHistory);
WoE_ClearHistory(In := _rt5.Q, out := Systemcontrolvars.control.b_ClearHistory); // WriteOnEdge

// NETWORK 6
_rt6(CLK := ExtControlVars.control.b_EMstop);
WoE_EMstop(In := _rt6.Q, out := SystemControlVars.control.b_EMstop); // WriteOnEdge

// NETWORK 7
_rt7(CLK := ExtControlVars.control.b_startDeHum);
WoE_DehumStart(In := _rt7.Q, out := SystemControlVars.control.b_startDeHum); // WriteOnEdge

// NETWORK 8
_rt8(CLK := ExtControlVars.control.b_Reset);
WoE_Reset(In := _rt8.Q, out := Systemcontrolvars.control.b_Reset); // WriteOnEdge
END_ACTION

METHOD RestoreDefaults
VAR_IN_OUT
	defaults 		: ST_Softsettings;
	softsettings	: ST_Softsettings;
END_VAR
IF memcmp(pBuf1 := ADR(defaults), pBuf2:= ADR(softsettings), n:= SIZEOF(defaults)) <> 0 THEN
	softsettings := defaults;
END_IF
END_METHOD

METHOD StoreDefaults : BOOL
VAR_IN_OUT
	defaults 		: ST_Softsettings;
	softsettings	: ST_Softsettings;
END_VAR
StoreDefaults := FALSE;

IF memcmp(pBuf1 := ADR(defaults), pBuf2:= ADR(softsettings), n:= SIZEOF(defaults)) <> 0 THEN
	defaults := softsettings;
ELSE
	StoreDefaults := TRUE;
END_IF
END_METHOD

END_FUNCTION_BLOCK

// ---- POUs/Functions-FBs-Programs/_generalFunctions/WriteOnEdge.TcPOU
FUNCTION_BLOCK WriteOnEdge
VAR_INPUT
	In	: BOOL;
END_VAR

VAR_IN_OUT
	out	:	BOOL;
END_VAR

VAR
	Ftrig	:	f_trig;
	Rtrig	:	r_trig;
END_VAR

//this function block writes the input value to the output, but only when the input changes (falling or rising).
//When no edge detection happens, the output value remains untouched, allowing for parallel input values to 1 output.
//Pair with R_trig on the input for pulse output on input rising edge.

Ftrig(clk := in);
Rtrig(clk := in);

IF (Ftrig.Q OR Rtrig.Q) THEN
	out := in;
END_IF

END_FUNCTION_BLOCK

// ---- POUs/MonitoringControl/IoT/RestComOpenremote.TcPOU
FUNCTION_BLOCK RestComOpenremote
VAR_INPUT
	UpdateConfiguration	:	BOOL;
END_VAR

VAR_OUTPUT
	ConfigurationDone	:	BOOL;
END_VAR
VAR
	CreditLoad			: INT;
	bEnable			:	BOOL := TRUE;
	Connectiontimer		:	ton := (PT := T#30S);
	timevalue	:	TIME;
	WriteConfigsToDisk	:	BOOL;
END_VAR

VAR //HTTP client items
	HTTPConnectionSTate		:	eConnectionState;
    httpClient     			: FB_IotHttpClient;
    sBearerAccessToken 	: STRING(5000);
END_VAR

VAR //Asset JSON parser items
	AssetfbJson     : 	FB_JsonDomParser;
    AssetjsonDoc   	: 	SJsonValue;
	AssetJsonDocTxt	:	STRING(50000);
	sAssetURI	 	: 	STRING(80) := '/api/master/asset/5WGb8fQx2n68yDmW4rYh9B';
END_VAR

VAR //Gateway connection JSON parser items
	GWConnfbJson     	: 	FB_JsonDomParser;
    GWConnjsonDoc   	: 	SJsonValue;
	sGWConnURI	 		: 	STRING(80) := '/api/master/gateway/connection/master';

	PeriodicFBJson		:	FB_JsonDomParser;
	PeriodicRoot		:	Sjsonvalue;
	PeriodicProp		:	SjsonValue;
	PeriodicSJsonIterator :	sjsonAIterator;
	
	OnChangeFBJson		:	FB_JsonDomParser;
	OnChangeRoot		:	Sjsonvalue;
	OnChangeProp		:	SjsonValue;
	OnChangeSJsonIterator :	sjsonAIterator;
	
	ExcludeFBJson		:	FB_JsonDomParser;
	ExcludeRoot		:	Sjsonvalue;
	ExcludeProp		:	SjsonValue;
	ExcludeSJsonIterator :	sjsonAIterator;
END_VAR


VAR
	state	:	UINT;
	Index	:	UINT;
	b_test	:	BOOL;
END_VAR

VAR_IN_OUT CONSTANT
	{ attribute 'TcHmiSymbol.Hide' }
	monitor							: ST_System_Monitor;
END_VAR

VAR_IN_OUT 
	HMILogData						: ARRAY [1..2000] OF ST_IoTDataHMI;
	controlvars						: ST_ExtController_get;
	st_params						: ST_IOT_params;
	IOTCredits						: ST_IotData_credits;
END_VAR

VAR
    // ---- OAuth2 config ----
    sHost        : STRING(255) := '10.4.0.41';
    nPort        : UINT := 443;
    sClientId    : STRING(80) := 'utilities';
    sClientSecret: STRING(80) := 'VcbYh6xIxRYAjYR8bkKyHZlxOCwJTkmD';
END_VAR

HTTPClient.sHostName							:= sHost;
	HTTPClient.nHostPort							:= nPort;
	HTTPClient.bKeepAlive 							:= TRUE;
	HTTPClient.stTLS.bNoServerCertCheck				:= TRUE;
	HTTPClient.stTLS.sCA							:= 'c:\PLCUtility\rootCA.pem'; 
	HTTPClient.tConnectionTimeout					:= T#1M;
	
IF bEnable THEN
	Connectiontimer(in := HTTPConnectionSTate = eConnectionState.authorization_declined);

	IF NOT Connectiontimer.Q THEN
		HTTPClient.Execute();
		Authenticate();
	ELSE
		HttpClient.Disconnect();
	END_IF

	CASE state OF
	0:
		IF UpdateConfiguration THEN
			ConfigurationDone := FALSE;
			state := 1;
		END_IF
	1:
		IF PrepareAssetConfig() THEN
			IOTCredits.TotalCredits := GetLoggingBudget();
			state := 2;
		END_IF
	
	2:
		IF PrepareGWConnConfig() THEN
			state := 3;
			IOTCredits.UsedCredits := 0;
		END_IF
	3:
		
		FOR Index := 1 TO SIZEOF(HMILogData)/SIZEOF(HMILogData[1])-1 DO
			IF HMILogData[Index].LogType > eLogType.none THEN
				CreditLoad := SEL(HMILogData[Index].LogType = 0, TO_INT(HMILogData[Index].LogType) + (3 - TO_INT(HMILogData[Index].LogInterval)), 0 );
				IOTCredits.UsedCredits := IOTCredits.UsedCredits + CreditLoad;
				IF HMILogData[Index].Unit = '' THEN
					AddAttributeToAsset(HMILogData[Index].Label, e_ORAttributeType.text, (NOT HMILogData[Index].b_IOTWriteAllowed), '');
				ELSE
					AddAttributeToAsset(HMILogData[Index].Label, e_ORAttributeType.number, (NOT HMILogData[Index].b_IOTWriteAllowed), HMILogData[Index].Unit);
				END_IF
		
				AddAttributeToGWConnConfig(HMILogData[Index].Label, HMILogData[Index].LogInterval, HMILogData[Index].Logtype);
			ELSE
				AssetFBJson.RemoveMemberByName(AssetjsonDoc, HMILogData[Index].Label, TRUE);
				//RemoveAttributeFromAssetConfig(HMILogData[Index].Label);
			END_IF
		END_FOR
		
		IOTCredits.RemainingCredits := IOTCredits.TotalCredits - IOTCredits.UsedCredits;

		state := SEL(WriteConfigsToDisk, 4, 6);	
		b_test := TRUE;
		
	4:
		IF PushAssetData() THEN
			state := 5;
			b_test := TRUE;
		END_IF

	5:
		IF PushGWConnConfig() THEN
			//clear all json parsers to free up router memory
			GWConnfbJson.NewDocument();
			AssetfbJson.NewDocument();
			PeriodicFBJson.NewDocument();
			OnChangeFBJson.NewDocument();
			ExcludeFBJson.NewDocument();
			
			ConfigurationDone	:= TRUE;
			state := 0;
		END_IF
		
	6:
		AssetfbJson.SaveDocumentToFile('C:\PLCUtility\testAssetConfig.txt', b_test);
		IF NOT b_test THEN
			state := 7;
			b_test := TRUE;
		END_IF
	7:
		GWConnfbJson.SaveDocumentToFile('C:\PLCUtility\testGWConfig.txt', b_test);
		IF NOT b_test THEN
			state := 4;
		END_IF
	END_CASE	
ELSE
	HTTPConnectionSTate := eConnectionState.disconnected;
	HttpClient.Disconnect();
END_IF

METHOD AddAttributeToAsset : BOOL
VAR_INPUT
	sAttributeName			:	STRING;
	eAttributeType			:	e_ORAttributeType;
	bReadOnly				:	BOOL;
	sUnit					:	STRING;
END_VAR

VAR_INST
	Initialized			:	BOOL;
	Attributefbjson		:	FB_JsonDomParser;
END_VAR
VAR_inst
	Attribute			:	SJsonValue;
	MetaJson			:	SJsonValue;
	AttributeSet		:	Sjsonvalue;
	sMetastring			:	STRING(1000);
	NewAttribute		:	STRING(5000);
END_VAR

VAR
	UnitA	:	STRING;
	UnitB	:	STRING;
	UnitC	:	STRING;
	UnitD	:	String;
	Separator : STRING := ' ';
	SpaceIndex	:	INT;
END_VAR
IF NOT Initialized THEN //initialize meta subjson once. 
	Attribute := Attributefbjson.NewDocument();
	Attributefbjson.AddBoolMember(Attribute, 'ruleState', TRUE);
	Attributefbjson.AddBoolMember(Attribute, 'accessRestrictedRead', TRUE);
	Attributefbjson.AddBoolMember(Attribute, 'storeDataPoints', TRUE);
	Attributefbjson.AddBoolMember(Attribute, 'accessPublicRead', TRUE);
	Attributefbjson.AddBoolMember(Attribute, 'readOnly', TRUE);
	sMetastring := Attributefbjson.GetDocument();
	Initialized := TRUE;
END_IF


Attribute := Assetfbjson.FindMember(AssetJsonDoc, sAttributeName);
IF Attribute <> 0 THEN //attribute already exists, but do update meta data.
	MetaJson := AssetFBJson.FindMember(Attribute, 'meta');
	IF MetaJson = 0 THEN
		MetaJson := Assetfbjson.AddJsonMember(Attribute, 'meta', sMetastring);
	END_IF
	
	AttributeSet := AssetFBJson.FindMember(MetaJson, 'readOnly');
	IF AttributeSet = 0 THEN
		AssetFBJson.AddBoolMember(MetaJson, 'readOnly', bReadOnly);
	ELSE
		AssetFBJson.SetBool(AttributeSet, bReadOnly);
	END_IF
	
	
	AssetFBJson.RemoveMemberByName(MetaJson, 'units', TRUE);
	IF sUnit <> '' THEN
		AttributeSet := AssetFBJson.AddArrayMember(MetaJson, 'units', 0);
		SpaceIndex := find(sUnit,' ');
		IF spaceIndex = 0 THEN
			AssetFBJson.PushbackStringValue(AttributeSet, sUnit);
		ELSE
			UnitA := left(sUnit, SpaceIndex-1);
			AssetFBJson.PushbackStringValue(AttributeSet, UnitA);
			Unitb := right(sUnit, len(sUnit)-SpaceIndex);
			SpaceIndex := find(Unitb, ' ');
			IF spaceIndex = 0 THEN
				AssetFBJson.PushbackStringValue(AttributeSet, Unitb);
			ELSE
				UnitC := right(Unitb, len(unitb)-SpaceIndex);
				Unitb := left(Unitb, SpaceIndex-1);
				AssetFBJson.PushbackStringValue(AttributeSet, UnitB);
				AssetFBJson.PushbackStringValue(AttributeSet, UnitC);
			END_IF
		END_IF
	END_IF
	

ELSE //attribute doesn't exist, create attribute and add.
	Attribute := Attributefbjson.NewDocument();
	Attributefbjson.AddStringMember(Attribute, 'name', sAttributeName);
	
	CASE eAttributeType OF
		e_ORAttributeType.integer	: Attributefbjson.AddStringMember(Attribute, 'type', 'integer');
		e_ORAttributeType.number	: Attributefbjson.AddStringMember(Attribute, 'type', 'number');
		e_ORAttributeType.text	: Attributefbjson.AddStringMember(Attribute, 'type', 'text');
		e_ORAttributeType.JSON	: Attributefbjson.AddStringMember(Attribute, 'type', 'JSON');
	END_CASE
	
	MetaJson := Assetfbjson.AddJsonMember(Attribute, 'meta', sMetastring);
	
	IF sUnit <> '' THEN
		AttributeSet := AssetFBJson.AddArrayMember(MetaJson, 'units', 0);
//		AssetFBJson.PushbackStringValue(AttributeSet, 'test4');
//		AssetFBJson.PushbackStringValue(AttributeSet, 'test5');
//		AssetFBJson.PushbackStringValue(AttributeSet, 'test6');
		AssetFBJson.setArray(AttributeSet, 0);
		SpaceIndex := find(sUnit, ' ');
		IF spaceIndex = 0 THEN
			AssetFBJson.PushbackStringValue(AttributeSet, sUnit);
		ELSE
			UnitA := left(sUnit, SpaceIndex-1);
			AssetFBJson.PushbackStringValue(AttributeSet, UnitA);
			Unitb := right(sUnit,  len(sUnit)-SpaceIndex);
			SpaceIndex := find(Unitb, ' ');
			IF spaceIndex = 0 THEN
				AssetFBJson.PushbackStringValue(AttributeSet, Unitb);
			ELSE
				
				UnitC := right(Unitb,  len(unitb)-SpaceIndex);
				Unitb := left(Unitb, SpaceIndex-1);
				AssetFBJson.PushbackStringValue(AttributeSet, UnitB);
				SpaceIndex := find(Unitc, ' ');
				IF spaceIndex = 0 THEN
					AssetFBJson.PushbackStringValue(AttributeSet, Unitc);
				ELSE
					UnitD := right(Unitc,  len(unitc)-SpaceIndex);
					Unitc := left(Unitc, SpaceIndex-1);
					AssetFBJson.PushbackStringValue(AttributeSet, UnitC);
					AssetFBJson.PushbackStringValue(AttributeSet, UnitD);
				END_IF
			END_IF
		END_IF
	END_IF
	
	AttributeSet := AssetFBJson.FindMember(MetaJson, 'readOnly');
	AssetFBJson.SetBool(AttributeSet, bReadOnly);
	Attributefbjson.CopyDocument(NewAttribute, SIZEOF(NewAttribute));
	Assetfbjson.AddJsonMember(AssetJsonDoc, sAttributeName, NewAttribute);
END_IF
END_METHOD

METHOD AddAttributeToGWConnConfig : BOOL
VAR_INPUT
	sAttributeName			:	STRING;
	eLogInterval			:	eUpdate;
	e_LogType				:	eLogType;
END_VAR

VAR
	NewAttribute		:	STRING(5000);
END_VAR

IF e_LogType = eLogType.cloud THEN
	NewAttribute := CreateMatcherItem(sAttributeName);
	
	//daily updates merged to onchange for now. The value will just be only changed daily via MQTT.
	IF eLogInterval = eUpdate.Onchange OR eLogInterval = eUpdate.Daily THEN
		GWConnfbJson.pushbackJsonValue(OnchangeProp, NewAttribute);
	ELSE
		GWConnfbJson.pushbackJsonValue(PeriodicProp, NewAttribute);
	END_IF
	
ELSIF e_LogType = eLogType.nuc THEN
	GWConnFBJSON.PushbackStringValue(ExcludeProp, sAttributeName);
END_IF
END_METHOD

METHOD Authenticate : BOOL
VAR_INPUT
	
END_VAR

VAR_INST
	eState	:	INT;
	TimeoutDone	: TON	:= ( Pt := T#30S);
	
	fbReqToken   : FB_IotHttpRequest;
    fbReqApi     : FB_IotHttpRequest;

    fbHdrToken   : FB_IotHttpHeaderFieldMap;
    fbHdrApi     : FB_IotHttpHeaderFieldMap;


    // ---- Payload / response buffers ----
    sFormBody    : STRING(512);
	sJsonDocContent	:	STRING(4096);
	SBearerSubstring	:	STRING(80);

    // ---- JSON parse (Tc3_JsonXml) ----
    fbJson       : FB_JsonDomParser;
    jsonDoc      : SJsonValue;
    jsonAccess   : SJsonValue;
	jsonToken	:	SJsonValue;
	
	rtrigConnected : r_trig;
	InitConnection	:	R_trig;
	
	bEnableb	:	Bool;
END_VAR
TimeoutDone();

rtrigConnected(clk := HTTPClient.bConnected);
IF rtrigConnected.Q THEN
	HTTPConnectionSTate := eConnectionState.connected;
END_IF

InitConnection(clk := bEnable AND HTTPConnectionSTate = eConnectionState.disconnected);
	
	CASE eState OF
		0: // Configure client & start token request
			IF InitConnection.q OR TimeoutDone.Q THEN
				TimeoutDone.IN := FALSE;
		
				// Build x-www-form-urlencoded body for client_credentials
				sFormBody := CONCAT('grant_type=client_credentials&client_id=', sClientId);
				sFormBody := CONCAT(sFormBody, '&client_secret=');
				sFormBody := CONCAT(sFormBody, sClientSecret);
				
				// Headers
				fbHdrToken.AddField(sField := 'Content-Type', sValue := 'application/x-www-form-urlencoded', bAppendValue := FALSE);
				fbHdrToken.AddField(sField := 'Accept',       sValue := 'application/json',              bAppendValue := FALSE);
		
				// Send POST with body
				fbReqToken.SendRequest(
					sUri := '/auth/realms/master/protocol/openid-connect/token',
					fbClient      := HTTPClient,
					eRequestType  := ETcIotHttpRequestType.HTTP_POST,
					pContent      := ADR(sFormBody),
					nContentSize  := LEN(sFormBody),
					fbHeader      := fbHdrToken
				);
		
				eState := 1;
			END_IF
		
		1: // Wait for token response
			IF NOT fbReqToken.bBusy THEN
				IF fbReqToken.bError THEN
					eState := -1;
				ELSE
					jsonDoc := fbReqToken.GetJsonDomContent(fbJson := fbJson);
					jsonAccess := fbJson.FindMember(v := jsonDoc, member := 'access_token');
					IF jsonAccess <> 0 THEN
						fbJson.CopyString(jsonAccess, sBearerAccessToken, SIZEOF(sBearerAccessToken));
						SBearerSubstring := 'Bearer ';
						concat2(ADR(SBearerSubstring), ADR(sBearerAccessToken), ADR(sBearerAccessToken), SIZEOF(sBearerAccessToken));
						TimeoutDone.IN := TRUE;
						HTTPConnectionSTate := eConnectionState.authorized;
						eState := 0;
					ELSE
						eState := -2;
					END_IF
				END_IF
			END_IF
		
		-1, -2:
			HTTPConnectionSTate := eConnectionState.authorization_declined;
			
		END_CASE
END_METHOD

METHOD CreateMatcherItem : String(1000)
VAR_INPUT
	sVarname	:	String(255);
END_VAR

VAR_INST
	MatcherFBJson	:	FB_JsonDomParser;
	NewItemroot		: 	SjsonValue;
	JsonProp		:	SjsonValue;
	Initialized		:	BOOL;
END_VAR

//creating the base structure is only done once.
IF NOT Initialized THEN
	NewItemroot := MatcherFBJson.NewDocument();
	JsonProp := MatcherFBJson.AddJsonMember(NewItemroot, 'name', '');
	MatcherFBJson.AddStringMember(JsonProp, 'predicateType', 'string');
	MatcherFBJson.AddStringMember(JsonProp, 'match', 'EXACT');
	MatcherFBJson.AddBoolMember(JsonProp, 'caseSensitive', TRUE);
	MatcherFBJson.AddBoolMember(JsonProp, 'negate', FALSE);
	MatcherFBJson.AddBoolMember(NewItemroot, 'negated', FALSE);
	JsonProp := MatcherFBJson.AddStringMember(JsonProp, 'value', '');
END_IF

//UpdateVarname as required
JsonProp := MatcherFBJson.SetString(JsonProp, sVarname);
//export item as string and return to output var.
MatcherFBJson.CopyDocument(CreateMatcherItem, SIZEOF(CreateMatcherItem));
END_METHOD

METHOD GetAssetData : BOOL
VAR_INST
    fbReqApi     : FB_IotHttpRequest;
    fbHdrApi     : FB_IotHttpHeaderFieldMap;
	eState		:	INT;
	bOk	:	BOOL;
	StartRead		:	R_trig;
	WaitForData		:	BOOL;
END_VAR
IF NOT WaitForData THEN	
	fbHdrApi.AddField(sField := 'Accept', sValue := 'application/json', bAppendValue := FALSE);
	fbHdrApi.AddField(sField := 'Authorization', sValue := sBearerAccessToken, bAppendValue := FALSE);
	
	fbReqApi.SendRequest(
		sUri := sAssetURI,
		fbClient      := HTTPClient,
		eRequestType  := ETcIotHttpRequestType.HTTP_GET,
		pContent      := 0,
		nContentSize  := 0,
		fbHeader      := fbHdrApi
	);
	
	WaitForData := TRUE;
END_IF

IF NOT fbReqApi.bBusy THEN
   IF NOT fbReqApi.bError THEN
	   AssetJsonDoc := fbReqApi.GetJsonDomContent(AssetfbJson);
	   GetAssetData := TRUE;
	ELSE
		GetAssetData := FALSE;
	END_IF
	
	WaitForData := FALSE;
END_IF
END_METHOD

METHOD GetGWConnConfig : BOOL
VAR_INST
    fbReqApi     : FB_IotHttpRequest;
    fbHdrApi     : FB_IotHttpHeaderFieldMap;
	eState		:	udINT;
	bOk	:	BOOL;
	loadDone, b_test	:	Bool;
	StartRead		:	R_trig;
	WaitForData		:	BOOL;
	
	JsonListElement	:	SJsonvalue;
	iterator		:	SJsonAIterator;
	iteratorEnd		:	SJSonAITerator;
	testA			:	STRING [20000];
	testB			:	STRING [20000];
	size	:	UDINT;
	isarr	:	BOOL;
	isjson	:	BOOL;
	membername : STRING(255);
END_VAR
IF NOT WaitForData THEN	
	fbHdrApi.AddField(sField := 'Accept', sValue := 'application/json', bAppendValue := FALSE);
	fbHdrApi.AddField(sField := 'Authorization', sValue := sBearerAccessToken, bAppendValue := FALSE);
	
	fbReqApi.SendRequest(
		sUri := sGWConnURI,
		fbClient      := HTTPClient,
		eRequestType  := ETcIotHttpRequestType.HTTP_GET,
		pContent      := 0,
		nContentSize  := 0,
		fbHeader      := fbHdrApi
	);
	
	WaitForData := TRUE;
END_IF
	
IF NOT fbReqApi.bBusy THEN
   IF NOT fbReqApi.bError THEN
	   GWConnjsonDoc 	:= fbReqApi.GetJsonDomContent(GWConnfbJson);
	   IF WriteConfigsToDisk THEN
		   LoadDone := TRUE;
		   b_test := TRUE;
		ELSE
			GetGWConnConfig := TRUE;
		END_IF
	ELSE
		GetGWConnConfig := FALSE;
	END_IF
	
	WaitForData := FALSE;
END_IF

IF loadDone THEN
	GWConnfbJson.SaveDocumentToFile('C:\PLCUtility\testGWConfig_orig.txt', b_test);
	IF NOT b_test THEN
		loadDone := FALSE;
		GetGWConnConfig := TRUE;
	END_IF
END_IF
END_METHOD

METHOD GetLoggingBudget : DINT
VAR_INPUT
END_VAR

VAR_INST
	Attribute			:	SJsonValue;
END_VAR
Attribute := Assetfbjson.FindMemberPath(AssetJsonDoc, 'W1/value/monitoringBudget' );
IF Attribute <> 0 THEN //attribute already exists, but do update meta data.
	GetLoggingBudget := TO_DINT(Assetfbjson.GetInt(Attribute));
ELSE //fallback value if no logging budget is read from the gateway
	GetLoggingBudget := st_params.DefaultLoggingBudget;
END_IF
END_METHOD

METHOD HTTPGetData : BOOL
VAR_IN_OUT
	sURI			:	STRING(1000);
	FBJSon			:	FB_JsonDomParser;
	JsonDoc			:	SJSonValue;
END_VAR

VAR_INST
    fbReqApi     : FB_IotHttpRequest;
    fbHdrApi     : FB_IotHttpHeaderFieldMap;
	WaitForData		:	BOOL;
END_VAR
IF NOT WaitForData THEN	
	fbHdrApi.AddField(sField := 'Accept', sValue := 'application/json', bAppendValue := FALSE);
	fbHdrApi.AddField(sField := 'Authorization', sValue := sBearerAccessToken, bAppendValue := FALSE);
	
	fbReqApi.SendRequest(
		sUri 			:= sURI,
		fbClient      	:= HTTPClient,
		eRequestType  	:= ETcIotHttpRequestType.HTTP_GET,
		pContent      	:= 0,
		nContentSize  	:= 0,
		fbHeader      	:= fbHdrApi
	);
	
	WaitForData := TRUE;
END_IF

HTTPGetData := FALSE;

IF NOT fbReqApi.bBusy THEN
   IF NOT fbReqApi.bError THEN
	   JsonDoc := fbReqApi.GetJsonDomContent(FBJSon);
	   HTTPGetData := TRUE;
	END_IF
END_IF
END_METHOD

METHOD PrepareAssetConfig : BOOL
VAR_INPUT
END_VAR
PrepareAssetConfig := FALSE;
//IF HTTPGetData(sURI := sAssetURI, fbjson := AssetfbJson, Jsondoc := AssetJsonDoc) THEN
IF GetAssetData() THEN
	AssetjsonDoc := AssetFBJson.FindMember(AssetjsonDoc, 'attributes');
	PrepareAssetConfig := TRUE;
END_IF
END_METHOD

METHOD PrepareGWConnConfig : BOOL
VAR_inst
	JsonIterator		:	SJsonAIterator;
	JsonIteratorEnd		:	SJsonAIterator;
	JsonValue, ArrayValue			:	SJsonVAlue;
	sPeriodicInterval	:	STRING;
	PeriodicInterval	:	TIME	:= T#134S;
	NrOfElements		:	UDINT;
	J					:	UDINT;
	Value				:	STRING;
	Tempstring			:	STRING(5000);
END_VAR

//VAR_IN_OUT
//	PeriodicFBJson		:	FB_JsonDomParser;
//	PeriodicRoot		:	Sjsonvalue;
//	PeriodicProp		:	SjsonValue;
//	PeriodicSJsonIterator :	sjsonAIterator;
	
//	OnChangeFBJson		:	FB_JsonDomParser;
//	OnChangeRoot		:	Sjsonvalue;
//	OnChangeProp		:	SjsonValue;
//	OnChangeSJsonIterator :	sjsonAIterator;
//END_VAR

VAR
	counter	:	UINT;
	NewAttribute		:	STRING(5000);
	Temp :	String;
	PeriodicMatcherTemplate		:	STRING(5000) 	:= '{"matcher": { "recursive": false, "realm": { "name": "master" }, "types": [ "EPU10" ], "attributes": { "operator": "OR", "items": [ { "name": { "predicateType": "string", "match": "EXACT", "caseSensitive": true, "value": "X1", "negate": false }, "negated": false }, { "name": { "predicateType": "string", "match": "EXACT", "caseSensitive": true, "value": "X9", "negate": false }, "negated": false }, { "name": { "predicateType": "string", "match": "EXACT", "caseSensitive": true, "value": "coolantPressure", "negate": false }, "negated": false }, { "name": { "predicateType": "string", "match": "EXACT", "caseSensitive": true, "value": "carbonMonoxidePpm", "negate": false }, "negated": false }, { "name": { "predicateType": "string", "match": "EXACT", "caseSensitive": true, "value": "upsStateOfCharge", "negate": false }, "negated": false }, { "name": { "predicateType": "string", "match": "EXACT", "caseSensitive": true, "value": "activePowerInverter", "negate": false }, "negated": false }, { "name": { "predicateType": "string", "match": "EXACT", "caseSensitive": true, "value": "activePowerOutput", "negate": false }, "negated": false }, { "name": { "predicateType": "string", "match": "EXACT", "caseSensitive": true, "value": "activePowerSetpoint", "negate": false }, "negated": false }, { "name": { "predicateType": "string", "match": "EXACT", "caseSensitive": true, "value": "ambientTemperature", "negate": false }, "negated": false }, { "name": { "predicateType": "string", "match": "EXACT", "caseSensitive": true, "value": "averageCellTemperature", "negate": false }, "negated": false }, { "name": { "predicateType": "string", "match": "EXACT", "caseSensitive": true, "value": "cabinetTemperature", "negate": false }, "negated": false }, { "name": { "predicateType": "string", "match": "EXACT", "caseSensitive": true, "value": "controlMode", "negate": false }, "negated": false }, { "name": { "predicateType": "string", "match": "EXACT", "caseSensitive": true, "value": "coolantTemperature", "negate": false }, "negated": false }, { "name": { "predicateType": "string", "match": "EXACT", "caseSensitive": true, "value": "cycleCount", "negate": false }, "negated": false }, { "name": { "predicateType": "string", "match": "EXACT", "caseSensitive": true, "value": "gridFilterTemperature", "negate": false }, "negated": false }, { "name": { "predicateType": "string", "match": "EXACT", "caseSensitive": true, "value": "hardwareConfiguration", "negate": false }, "negated": false }, { "name": { "predicateType": "string", "match": "EXACT", "caseSensitive": true, "value": "inverterTemperature", "negate": false }, "negated": false }, { "name": { "predicateType": "string", "match": "EXACT", "caseSensitive": true, "value": "loadPercentage", "negate": false }, "negated": false }, { "name": { "predicateType": "string", "match": "EXACT", "caseSensitive": true, "value": "location", "negate": false }, "negated": false }, { "name": { "predicateType": "string", "match": "EXACT", "caseSensitive": true, "value": "averageCellTemperature", "negate": false }, "negated": false }, { "name": { "predicateType": "string", "match": "EXACT", "caseSensitive": true, "value": "productionDate", "negate": false }, "negated": false }, { "name": { "predicateType": "string", "match": "EXACT", "caseSensitive": true, "value": "reactivePowerInverter", "negate": false }, "negated": false }, { "name": { "predicateType": "string", "match": "EXACT", "caseSensitive": true, "value": "relHumCabinet", "negate": false }, "negated": false }, { "name": { "predicateType": "string", "match": "EXACT", "caseSensitive": true, "value": "serialNumber", "negate": false }, "negated": false }, { "name": { "predicateType": "string", "match": "EXACT", "caseSensitive": true, "value": "stateOfCharge", "negate": false }, "negated": false }, { "name": { "predicateType": "string", "match": "EXACT", "caseSensitive": true, "value": "stateOfHealth", "negate": false }, "negated": false }, { "name": { "predicateType": "string", "match": "EXACT", "caseSensitive": true, "value": "throttlingPercentage", "negate": false }, "negated": false }, { "name": { "predicateType": "string", "match": "EXACT", "caseSensitive": true, "value": "totalEnergytoBattery", "negate": false }, "negated": false }, { "name": { "predicateType": "string", "match": "EXACT", "caseSensitive": true, "value": "totalEnergyFromBattery", "negate": false }, "negated": false }, { "name": { "predicateType": "string", "match": "EXACT", "caseSensitive": true, "value": "zeropointPowerload", "negate": false }, "negated": false } ] }, "limit": 0 }}';
	OnchangeMatcherTemplate 	: 	STRING(1000)	:='{ "matcher": { "recursive": false, "realm": { "name": "master" }, "types": [ "EPU10" ], "attributes": { "operator": "OR", "items": [ { "name": { "predicateType": "string", "match": "EXACT", "caseSensitive": true, "value": "operatingState", "negate": false }, "negated": false }, { "name": { "predicateType": "string", "match": "EXACT", "caseSensitive": true, "value": "urgentMessages", "negate": false }, "negated": false } ] }, "limit": 0 }, "valueChange": true, "durationParsedMillis": null}';
	skipAlwaysTemplate			:	STRING			:=	'{"skipAlways": true}';
	ExcludeAttributeTemplate 	: 	STRING(1500)	:=	'{"excludeAttributeMeta":{"*":["accessRestrictedWrite","accessPublicRead","accessPublicWrite","attributeLinks"]},"addAttributeMeta":{"*":{"accessPublicWrite":false,"accessPublicRead":false,"readOnly":true}},"accessPublicRead":false,"excludeAttributes":["availableEnergyCapacity","clientAbbreviation","currentDcCoupling","currentL1InputField","currentL1OutputField","currentL1Psb","currentL2InputField","currentL2OutputField","currentL2Psb","currentL3InputField","currentL3OutputField","currentL3Psb","currentNInputField","currentNOutputField","currentNPsb","dcLinkCurrent","dcLinkVoltage","frequency","idleChargePower","inverterAcCurrent","limitMaxPowerSetpoint","limitMinPowerSetpoint","lineVoltageL1L2","lineVoltageL2L3","lineVoltageL3L1","machineDescription","maxSocReserve","minSocReserve","model","peakShaveMax","peakShaveMin","pfL1","pfL2","pfL3","phaseVoltageL1","phaseVoltageL2","phaseVoltageL3","plcConnected","powerDcCoupling","reactivePowerInput","reactivePowerOutput","reactivePowerSetpoint","setOperation","shutdownCommand","shutdownReply","socTarget","transformerTemperature","voltageLL","voltageLN","X10","X11","X12","X13","X14","X15","X2","X3","X4","X5","X6","X7","X8"]}';
END_VAR
PrepareGWConnConfig := false;


//if HTTPGetData(sURI := sGWConnURI, fbjson := GWConnfbJson, Jsondoc := GWConnjsonDoc) then
if GetGWConnConfig() then
	//Removes existing gateway filters from json, updates interval timer to current setting, prepares Jsonpointers for to allow adding new config
	
	PeriodicRoot := GWConnfbJson.GetDocumentRoot();
	PeriodicProp := GWConnfbJson.FindMember(PeriodicRoot, 'attributeFilters');
	
	_ReturnLabel: 
	//Remove matcher configs if they contain the type definition for ePU10. 
	jsonIterator          := GWConnfbJson.ArrayBegin(PeriodicProp);
	jsonIteratorEnd       := GWConnfbJson.ArrayEnd(PeriodicProp);
	WHILE jsonIterator <> jsonIteratorEnd DO
	  jsonValue           := GWConnfbJson.GetArrayValue(jsonIterator);
	  jsonValue			  := GWConnfbJson.FindMemberPath(jsonValue, 'matcher/types');
	  IF jsonValue <> 0 THEN //types array exists
		NrOfElements := GWConnfbJson.GetArraySize(jsonValue);
		
		FOR j := 0 TO NrOfElements - 1 DO
			ArrayValue := GWConnfbJson.GetArrayValuebyidx(jsonValue, j);
			IF ArrayValue <> 0 THEN
				Value := GWConnfbJson.GetString(ArrayValue);
				IF Value = 'EPU10' THEN
					GWConnfbJson.RemoveArray(PeriodicProp, jsonIterator);
					JMP _ReturnLabel; //don't call nextArray if an element is removed, jump back to beginning of the loop
				END_IF
			END_IF
		END_FOR
	  ELSE
		jsonValue           := GWConnfbJson.GetArrayValue(jsonIterator);
		jsonValue			:= GWConnfbJson.FindMember(jsonValue, 'skipAlways');
	 	IF jsonValue <> 0 THEN //skipalways element exists, remove it to be re-added at the end
			GWConnfbJson.RemoveArray(PeriodicProp, jsonIterator);
			JMP _ReturnLabel; //don't call nextArray if an element is removed, jump back to beginning of the loop
		END_IF
	  END_IF
	  jsonIterator        := GWConnfbJson.NextArray(jsonIterator);
	END_WHILE
	
	PeriodicRoot := GWConnfbJson.PushbackJsonValue(PeriodicProp, PeriodicMatcherTemplate);
	IF PeriodicInterval >= T#1H THEN
		PeriodicInterval := T#59M59S;
	END_IF
	GWConnfbJson.AddIntMember(PeriodicRoot, 'durationParsedMillis', TIME_TO_DINT(PeriodicInterval));
	Temp := TIME_TO_STRING(PeriodicInterval);
	Temp :=  F_ToUCase(Temp);
	temp := concat('PT', right(Temp, len(Temp)-2));
	
	GWConnfbJson.AddStringMember(PeriodicRoot, 'duration', Temp);	//update interval time to current setting
	
	OnchangeRoot := GWConnfbJson.PushbackJsonValue(PeriodicProp, OnchangeMatcherTemplate);
	GWConnfbJson.PushbackJsonValue(PeriodicProp, skipAlwaysTemplate);
	OnchangeProp := GWConnfbJson.FindMember(OnchangeRoot, 'matcher');
	OnchangeProp := GWConnfbJson.FindMember(OnchangeProp, 'attributes');
	OnchangeProp := GWConnfbJson.FindMember(OnchangeProp, 'items');
	
	PeriodicProp := GWConnfbJson.FindMember(PeriodicRoot, 'matcher');
	PeriodicProp := GWConnfbJson.FindMember(PeriodicProp, 'attributes');
	PeriodicProp := GWConnfbJson.FindMember(PeriodicProp, 'items');
	
	ExcludeRoot := GWConnfbJson.GetDocumentRoot();
	ExcludeRoot  := GWConnfbJson.FindMember(ExcludeRoot, 'assetSyncRules');
	GWConnfbJson.RemoveMemberByName(ExcludeRoot, 'EPU10', TRUE);
	ExcludeProp := GWConnfbJson.addjsonmember(ExcludeRoot, 'EPU10', ExcludeAttributeTemplate);
	ExcludeProp  := GWConnfbJson.FindMember(ExcludeProp, 'excludeAttributes');

	//ExcludeSJsonIterator  := GWConnfbJson.ArrayBegin(ExcludeProp);
	//GWConnFBJson.setArray(ExcludeProp, 0);
	
	PrepareGWConnConfig := True;
end_if
END_METHOD

METHOD PrepareGWConnConfig_OLD : BOOL
VAR_inst

	sPeriodicInterval	:	STRING;
	PeriodicInterval	:	TIME	:= T#134S;
END_VAR

//VAR_IN_OUT
//	PeriodicFBJson		:	FB_JsonDomParser;
//	PeriodicRoot		:	Sjsonvalue;
//	PeriodicProp		:	SjsonValue;
//	PeriodicSJsonIterator :	sjsonAIterator;
	
//	OnChangeFBJson		:	FB_JsonDomParser;
//	OnChangeRoot		:	Sjsonvalue;
//	OnChangeProp		:	SjsonValue;
//	OnChangeSJsonIterator :	sjsonAIterator;
//END_VAR

VAR
	counter	:	UINT;
	NewAttribute		:	STRING(5000);
END_VAR
PrepareGWConnConfig_OLD := FALSE;


//if HTTPGetData(sURI := sGWConnURI, fbjson := GWConnfbJson, Jsondoc := GWConnjsonDoc) then
if GetGWConnConfig() then
	//Removes existing gateway filters from json, updates interval timer to current setting, prepares Jsonpointers for to allow adding new config
	
	PeriodicRoot := GWConnfbJson.GetDocumentRoot();
	PeriodicProp := GWConnfbJson.FindMember(PeriodicRoot, 'attributeFilters');
	
	PeriodicSJsonIterator  := GWConnfbJson.ArrayBegin(PeriodicProp);	//get first array element (periodic matcher)
	OnchangeSJsonIterator  := GWConnfbJson.nextarray(PeriodicSJsonIterator);	//switch to second array element (onchange matcher)
	
	PeriodicProp := GWConnfbJson.FindMember(PeriodicRoot, 'duration');	//update interval time to current setting
	sPeriodicInterval := TIME_TO_STRING(PeriodicInterval);
	GWConnfbJson.SetString(PeriodicProp, sPeriodicInterval);
	
	PeriodicProp := GWConnfbJson.FindMember(PeriodicRoot, 'durationParsedMillis');
	GWConnfbJson.Setint(PeriodicProp, TIME_TO_DINT(PeriodicInterval));
	
	PeriodicRoot := GWConnfbJson.GetArrayValue(PeriodicSJsonIterator);	//get root sjsonvalue of periodic matcher
	PeriodicProp := GWConnfbJson.FindMember(PeriodicRoot, 'matcher');
	
	PeriodicProp := GWConnfbJson.FindMember(PeriodicProp, 'attributes');
	PeriodicProp := GWConnfbJson.FindMember(PeriodicProp, 'items');
	PeriodicSJsonIterator  := GWConnfbJson.ArrayBegin(PeriodicProp);
	GWConnfbJson.ClearArray(PeriodicProp, PeriodicSJsonIterator);	//Clear current matching list
	GWConnFBJson.setArray(PeriodicProp, 0);
	//Periodic matcher now initialized, new matching values can now be pushed with pushbackjsonvalue and creatematcheritem()
	
	//First add default items
	NewAttribute := CreateMatcherItem('X1');						GWConnFBJson.pushbackjsonvalue(PeriodicProp,NewAttribute);
	NewAttribute := CreateMatcherItem('X9');						GWConnFBJson.pushbackjsonvalue(PeriodicProp,NewAttribute);
	NewAttribute := CreateMatcherItem('coolantPressure');			GWConnFBJson.pushbackjsonvalue(PeriodicProp,NewAttribute);
	NewAttribute := CreateMatcherItem('carbonMonoxidePpm');			GWConnFBJson.pushbackjsonvalue(PeriodicProp,NewAttribute);
	NewAttribute := CreateMatcherItem('upsStateOfCharge');			GWConnFBJson.pushbackjsonvalue(PeriodicProp,NewAttribute);
	NewAttribute := CreateMatcherItem('activePowerInverter');		GWConnFBJson.pushbackjsonvalue(PeriodicProp,NewAttribute);
	NewAttribute := CreateMatcherItem('activePowerOutput');			GWConnFBJson.pushbackjsonvalue(PeriodicProp,NewAttribute);
	NewAttribute := CreateMatcherItem('activePowerSetpoint');		GWConnFBJson.pushbackjsonvalue(PeriodicProp,NewAttribute);
	NewAttribute := CreateMatcherItem('ambientTemperature');		GWConnFBJson.pushbackjsonvalue(PeriodicProp,NewAttribute);
	NewAttribute := CreateMatcherItem('averageCellTemperature');	GWConnFBJson.pushbackjsonvalue(PeriodicProp,NewAttribute);
	NewAttribute := CreateMatcherItem('cabinetTemperature');		GWConnFBJson.pushbackjsonvalue(PeriodicProp,NewAttribute);
	NewAttribute := CreateMatcherItem('controlMode');				GWConnFBJson.pushbackjsonvalue(PeriodicProp,NewAttribute);
	NewAttribute := CreateMatcherItem('coolantTemperature');		GWConnFBJson.pushbackjsonvalue(PeriodicProp,NewAttribute);
	NewAttribute := CreateMatcherItem('cycleCount');				GWConnFBJson.pushbackjsonvalue(PeriodicProp,NewAttribute);
	NewAttribute := CreateMatcherItem('gridFilterTemperature');		GWConnFBJson.pushbackjsonvalue(PeriodicProp,NewAttribute);
	NewAttribute := CreateMatcherItem('hardwareConfiguration');		GWConnFBJson.pushbackjsonvalue(PeriodicProp,NewAttribute);
	NewAttribute := CreateMatcherItem('inverterTemperature');		GWConnFBJson.pushbackjsonvalue(PeriodicProp,NewAttribute);
	NewAttribute := CreateMatcherItem('loadPercentage');			GWConnFBJson.pushbackjsonvalue(PeriodicProp,NewAttribute);
	NewAttribute := CreateMatcherItem('location');					GWConnFBJson.pushbackjsonvalue(PeriodicProp,NewAttribute);
	NewAttribute := CreateMatcherItem('averageCellTemperature');	GWConnFBJson.pushbackjsonvalue(PeriodicProp,NewAttribute);
	NewAttribute := CreateMatcherItem('productionDate');			GWConnFBJson.pushbackjsonvalue(PeriodicProp,NewAttribute);
	NewAttribute := CreateMatcherItem('reactivePowerInverter');		GWConnFBJson.pushbackjsonvalue(PeriodicProp,NewAttribute);
	NewAttribute := CreateMatcherItem('relHumCabinet');				GWConnFBJson.pushbackjsonvalue(PeriodicProp,NewAttribute);
	NewAttribute := CreateMatcherItem('serialNumber');				GWConnFBJson.pushbackjsonvalue(PeriodicProp,NewAttribute);
	NewAttribute := CreateMatcherItem('stateOfCharge');				GWConnFBJson.pushbackjsonvalue(PeriodicProp,NewAttribute);
	NewAttribute := CreateMatcherItem('stateOfHealth');				GWConnFBJson.pushbackjsonvalue(PeriodicProp,NewAttribute);
	NewAttribute := CreateMatcherItem('throttlingPercentage');		GWConnFBJson.pushbackjsonvalue(PeriodicProp,NewAttribute);
	NewAttribute := CreateMatcherItem('totalEnergytoBattery');		GWConnFBJson.pushbackjsonvalue(PeriodicProp,NewAttribute);
	NewAttribute := CreateMatcherItem('totalEnergyFromBattery');	GWConnFBJson.pushbackjsonvalue(PeriodicProp,NewAttribute);
	NewAttribute := CreateMatcherItem('zeropointPowerload');		GWConnFBJson.pushbackjsonvalue(PeriodicProp,NewAttribute);	
	
	
	OnchangeRoot := GWConnfbJson.GetArrayValue(OnchangeSJsonIterator);	//get root sjsonvalue of Onchange matcher
	OnchangeProp := GWConnfbJson.FindMember(OnchangeRoot, 'matcher');
	OnchangeProp := GWConnfbJson.FindMember(OnchangeProp, 'attributes');
	OnchangeProp := GWConnfbJson.FindMember(OnchangeProp, 'items');
	OnchangeSJsonIterator  := GWConnfbJson.ArrayBegin(OnchangeProp);
	GWConnfbJson.ClearArray(OnchangeProp, OnchangeSJsonIterator);	//Clear current matching list
	GWConnFBJson.setArray(OnchangeProp, 0);

	//onchange matcher now initialized, new matching values can now be pushed with pushbackjsonvalue and creatematcheritem()
	//First add default items
	NewAttribute := CreateMatcherItem('operatingState');
	GWConnFBJson.pushbackjsonvalue(OnchangeProp,NewAttribute);
	
	NewAttribute := CreateMatcherItem('urgentMessages');
	GWConnFBJson.pushbackjsonvalue(OnchangeProp,NewAttribute);
	
	
	ExcludeRoot := GWConnfbJson.GetDocumentRoot();
	ExcludeRoot  := GWConnfbJson.FindMember(ExcludeRoot, 'assetSyncRules');
	ExcludeProp  := GWConnfbJson.FindMember(ExcludeRoot, 'EPU10');
	IF ExcludeProp = 0 THEN
		ExcludeProp := GWConnfbJson.addjsonmember(ExcludeRoot, 'EPU10', '');
	END_IF
	
	ExcludeProp  := GWConnfbJson.FindMember(ExcludeProp, 'excludeAttributes');
	IF ExcludeProp = 0 THEN
		ExcludeProp := GWConnfbJson.addArraymember(ExcludeProp, 'excludeAttributes',0);
	END_IF
	
	ExcludeSJsonIterator  := GWConnfbJson.ArrayBegin(ExcludeProp);
	GWConnfbJson.ClearArray(ExcludeProp, ExcludeSJsonIterator);	//Clear current matching list
	GWConnFBJson.setArray(ExcludeProp, 0);
	
	PrepareGWConnConfig_OLD := TRUE;
end_if
END_METHOD

METHOD PushAssetData : BOOL
//VAR_INPUT
//	pdata	:	POINTER TO STRING;
//	nData	:	UDINT;
//END_VAR


VAR_INST
    fbReqApi     : FB_IotHttpRequest;
    fbHdrApi     : FB_IotHttpHeaderFieldMap;
	eState		:	INT;
	bOk	:	BOOL;
	StartRead		:	R_trig;
	WaitForData		:	BOOL;
END_VAR
IF NOT waitforData THEN	
	fbHdrApi.AddField(sField := 'Accept', sValue := 'application/json', bAppendValue := FALSE);
	fbHdrApi.AddField(sField := 'Authorization', sValue := sBearerAccessToken, bAppendValue := FALSE);
	fbHdrApi.AddField(sField := 'Content-Type', sValue := 'application/json', bAppendValue := FALSE);
	
	fbReqApi.SendJsonDomRequest(
		sUri := sAssetURI,
		fbClient      := HTTPClient,
		eRequestType  := ETcIotHttpRequestType.HTTP_PUT,
		fbJson := AssetfbJson,
		fbHeader      := fbHdrApi
	);
	
	WaitForData := TRUE;
END_IF
	
IF NOT fbReqApi.bBusy THEN
   IF NOT fbReqApi.bError THEN
	   PushAssetData := TRUE;
	ELSE
		PushAssetData := FALSE;
	END_IF
	
	WaitForData := FALSE;
END_IF
END_METHOD

METHOD PushGWConnConfig : BOOL
//VAR_INPUT
//	pdata	:	POINTER TO STRING;
//	nData	:	UDINT;
//END_VAR


VAR_INST
    fbReqApi     : FB_IotHttpRequest;
    fbHdrApi     : FB_IotHttpHeaderFieldMap;
	eState		:	INT;
	bOk	:	BOOL;
	StartRead		:	R_trig;
	WaitForData		:	BOOL;
	
	OutputData	:	STRING(1000);
END_VAR
IF NOT waitforData THEN	
	fbHdrApi.AddField(sField := 'Accept', sValue := 'application/json', bAppendValue := FALSE);
	fbHdrApi.AddField(sField := 'Authorization', sValue := sBearerAccessToken, bAppendValue := FALSE);
	fbHdrApi.AddField(sField := 'Content-Type', sValue := 'application/json', bAppendValue := FALSE);
	
	fbReqApi.SendJsonDomRequest(
		sUri := sGWConnURI,
		fbClient      := HTTPClient,
		eRequestType  := ETcIotHttpRequestType.HTTP_PUT,
		fbJson := GWConnfbJson,
		fbHeader      := fbHdrApi
	);
	
	WaitForData := TRUE;
END_IF
	
IF NOT fbReqApi.bBusy THEN
   //fbReqApi.GetContent(adr(OutputData), sizeof(OutputData), true);
   IF NOT fbReqApi.bError THEN
	   PushGWConnConfig := TRUE;
	ELSE
		PushGWConnConfig := FALSE;
	END_IF
	
	WaitForData := FALSE;
END_IF
END_METHOD

METHOD RemoveAttributeFromAssetConfig : BOOL
VAR_INPUT
	AttributeName	:	String;
END_VAR

VAR_INST
	Index	:	UInt;
END_VAR
END_METHOD

END_FUNCTION_BLOCK

// ---- POUs/MonitoringControl/IoT/MqttComOpenremote.TcPOU
PROGRAM MqttComOpenremote
VAR
	sStartShutdownCMD	: STRING;
	sEventMsg			: STRING(2000);
	eActiveMsg			: eSeverity; // range from 0 to 5. 0 = none, 1 info, ... 5 em shutdown
	productionDateString: STRING;
	bInitiateFirstTimeSend : BOOL;
	w_shutdown			: WORD; //0 = remain, 1 = shutdown request
	s_ShutdownFb		: STRING;
	rtrig_shutdownRequested		:	R_trig;
END_VAR

VAR
	timer1: profiler;
	testword : WORD;
	b_UpdateActive	: BOOL;

	// Function blocks
	fbMqttClient 					: FB_IotMqttClient;
	fbMessageQueue					: FB_IotMqttMessageQueue;
    fbMessage						: FB_IotMqttMessage;
	fbJsonWriter					: FB_JsonSaxWriter;
	fbJsonDataType					: FB_JsonReadWriteDataType;
	fbJson							: FB_JsonDomParser;
	// Internal Vars
	ConnectionState					: ETCIOTMQTTCLIENTSTATE;

	stAutoProvisioning				: ST_AutoProvisioning;
	stAutoProvClear					: ST_Autoprovisioning;
	i								: INT; // for loop index
	bSetParameter 					: BOOL := TRUE;
	bConnect 						: BOOL := TRUE;	


	bSubscribed						: BOOL;
	bIncommingMsg					: BOOL;
	{attribute 'TcEncoding':='UTF-8'}
	receivingTopic					: STRING(255);
	{attribute 'TcEncoding':='UTF-8'}
	sMessage						: STRING(255);
	sMessageEmpty					: STRING(255);
	//sMessageEmpty					: STRING(20000);
	{attribute 'TcEncoding':='UTF-8'}
	bSubscribedAutoProv				: BOOL;
	hrErrorOccurred 				: DINT; //Contains latest error message
	st_IotProps						: ST_IotProps;
	sTopic							: STRING;
	aPreviousValue					: ARRAY[1..20] OF STRING(2000); //Stores values for onChange trigger. Keep this array as long as the IoTMapping Case!!
	sSubscribtion					: STRING(255);
	sSubChecker						: STRING(255);
	
	//Settings
	fbSendFastMessageTimer			: TON := (PT:=T#15S); 
	fbSendSlowMessageTimer			: TON := (PT:=T#60S);
	fbDailyTimer					: TON := (PT:=T#1D); //used for daily reconnect, which also results in sending eUpdate.Daily messages
	fbConnectionTimer				: TON := (PT:=T#5S);
	iSizeIotMappingV1				: INT := 100;
	iSizeTotal						: INT  := 0;
	iSizeMax						: INT := 2000;
	sPubPrefix						: STRING  := 'master/plc/writeattributevalue/';
	sSubPrefix						: STRING  := 'master/plc/attributevalue/';  // only use attributevalue, this code does not process full /attribute/ message
	sAssetID						: STRING  := '/5WGb8fQx2n68yDmW4rYh9B';
	{attribute 'TcEncoding':='UTF-8'}
	autoProvSub						: STRING(255) := 'provisioning/device2/response';
	{attribute 'TcEncoding':='UTF-8'}
	autoProvPub						: STRING(255) := 'provisioning/device2/request';
	
	s_AutoProvMsg					: STRING(4010):= '{"type": "x509","cert": "-----BEGIN CERTIFICATE-----\nMIIFPTCCAyUCFDQ4u2+PTWiPgHVzlYHSt5SDqQoPMA0GCSqGSIb3DQEBCwUAMGMx\nCzAJBgNVBAYTAk5MMRMwEQYDVQQIDApTb21lLVN0YXRlMQ8wDQYDVQQHDAZBbG1l\nbG8xGzAZBgNVBAoMElZETCBFbmVyZ3kgU3lzdGVtczERMA8GA1UEAwwIVkVTIENB\nIDIwIBcNMjQwMzEzMTQxMDU4WhgPMjEyNDAyMTgxNDEwNThaMFExCzAJBgNVBAYT\nAk5MMRMwEQYDVQQIDApPdmVyaWpzc2VsMRswGQYDVQQKDBJWREwgRW5lcmd5IFN5\nc3RlbXMxEDAOBgNVBAMMB2RldmljZTIwggIiMA0GCSqGSIb3DQEBAQUAA4ICDwAw\nggIKAoICAQCiwnpUiyODuS5kLG+Zi7te7CUrHVIp+ZA39L/wISaBE7/z9MRjYxVK\notSnVWUyCt+pU3EHkC4X6SQz7vRuQET13L49LOYjUD/Gn4t87YD/Kj5r/9cj7Vf3\nxnI+1Kwh7BmajAtsB3wVZxe/RmCfO9D7SGors4gGI+RZAvV3U0hHFWHU6G2TCb+q\nJfp71xQJQUp4QW6USlSAC2d77BbXMyV+c1FYaoqJIInd5JgEK6WQpoZ4S+A8P7AO\n2rbMRsPMrvDAe7WpsbQNZnHfEgV7nEP6+19D0fum3q0fp68hrnzyvRJ90ShOS6Le\n+mdnd326RP6LzTd+mXgcAmHczJiiQ1iY+OtC9VySsylsfW2VngJQaYd+f88Sx/85\nQCOwp4oA5hrNDIfQU1JnRDoVcSnPIvyzpqrERig6IEtpgT2DG32VOgne47ut0H0r\nIE7mXlRXYmSkKTws2Iph2nKpwwSdcvtYY+DrmPgT3EE7jAP/OkMNr0afQFmvqaQ+\n2SbxiivPxUwJLXGccrBmV1J3A91JbNwVdhvD3Ab0Rf/O8yWN0yEJ5X5e1q+b7hwa\nfh04iF8BM+ofYNGu74CKDq4cSWoU431G86TW2EMus6W0BCcvh3O+jGDNQ6bzfqYq\nUq+It8m5WpWjsvZtmXROFeCAsGK45eKdRR72zXl4YOItXaVqUzCr2QIDAQABMA0G\nCSqGSIb3DQEBCwUAA4ICAQB7n0i/OYpdXb5fgRe2fQ9IFIfXF7K88rzKgh+B1SWP\nVqfp8l5uHQZO9+k2qFmUbPdvE+zSlOuS98/cEErLdUOJvMidIAAkJHSr2F8IoLoT\nJgHEhj/SD5EBWEgsWV/6GewwpCOW21dA3Y1pgANWOK7KxoWkcLRb5iykBe5z8AU7\n+LDPNVnhdy+GuFkpzvEUiYL8CSYDJT28o1Rs9+HxglUZ39faTCU82O1rGJ+l9L2a\nWU3vwI7vqDEzIFfEHn48+XUoZVXgq818a1pSaJil7pMZb0EYbJHDHQGvetL8gddc\n1Rcibmofu/ZBXoK1bxk7KgJ9lEjO4BoZZ0tK19APuxBjClIBm7oTnj87+/YJfBfk\nQMSzDe30u+TdHRKIWa4DckzFFTBQsNg8T+t9PbhS1kD1D0dECBzbllOnD2v6xbf+\nshnK5LWrgIoKVpocyTc46B4S0g9Drk2eDOtA3G3SH+IbT8wgeIxiqDNRHYFcHDjq\nAOQpB9xGhmsURHuv+l0gwMmi7/Ru5MXkVJrAplkFN/ShB961xzcfERn9dsgcP/75\nlHY7qglTN5gSh/QFime0JgV1Om2VantZXQUiQGsgFbMgivjV5qo57Y9T+xg5EKT8\nx2IR2GTsnK9H7Q0TNAeTGV0qcN6tIGpfQHe8f9o3LLq4QaHeR3JYhZhkiC6i+lnw\nAA==\n-----END CERTIFICATE-----\n-----BEGIN CERTIFICATE-----\nMIIFqTCCA5GgAwIBAgIUNrEQi2T7AK4cV+ePfFtr0IBVl6MwDQYJKoZIhvcNAQEL\nBQAwYzELMAkGA1UEBhMCTkwxEzARBgNVBAgMClNvbWUtU3RhdGUxDzANBgNVBAcM\nBkFsbWVsbzEbMBkGA1UECgwSVkRMIEVuZXJneSBTeXN0ZW1zMREwDwYDVQQDDAhW\nRVMgQ0EgMjAgFw0yNDAzMTMxNDEwNDlaGA8yMTI0MDIxODE0MTA0OVowYzELMAkG\nA1UEBhMCTkwxEzARBgNVBAgMClNvbWUtU3RhdGUxDzANBgNVBAcMBkFsbWVsbzEb\nMBkGA1UECgwSVkRMIEVuZXJneSBTeXN0ZW1zMREwDwYDVQQDDAhWRVMgQ0EgMjCC\nAiIwDQYJKoZIhvcNAQEBBQADggIPADCCAgoCggIBAJ2dmmFb3vcP92xgubb/DQBn\nrX1HV93mzthCntSKvTOsyIpZJQ35c8OyL35qq6nzLj/iDoGrQxC+zKghKzRB1HhO\nNg2DnXNNqzvug/m4PXao5w59D//VWP70mT6yfhgsFJKzJNi3EnPLiz41HP6/hLG0\nwudKpIK3j25Wm70FsWvw2z1icUDcyp7Ef7Ob4Koy7uOsDa5W8tZDlN3hDlU784T9\nzvlxTSvvK4uHz+Qi+1R6OVMoiBB6ZtXfQKSUrEHwNTXKjt51vR8bEdZamNUW5O8L\nl4yGenkySDEZdPvG43SZS1+CV5zSSiVCxSbFGSIO8c5ldkAUS/MMwxpIgXpf2xyS\nSstF6mebFl0Ij/EXybkh5tz8DWAsnSm6gRhaLhpdtgBZX4v43p47CRGY8DoeGzA6\ne2aFgtVQTDI3Gvr1nVQR7wkdQh0YzETy7vbBIy7HYXQw6pE/eskFSEEKFChxvkL7\nQHAcRp1RaXNOQM2uja/1h16HFxRFNd91BCdmUms64DuXAIBXteSt6bfINle4Znne\n2rUrTkvZw+6MMPVn44IrzgKbYv0bZEFPMtaLXNp1BPNMkzsNtAuLXLRm//9KA9ov\nGr/NMdO9j1e72/myYYD0+T165GTO5ZIS92jOkyb+REOAHz4R1Nb1eluehiJ0zVgK\nM78ki4Z+Z1nBxIkbByq3AgMBAAGjUzBRMB0GA1UdDgQWBBTKkYlzFWWdQk8jl6Wm\nkl+r4hoY8zAfBgNVHSMEGDAWgBTKkYlzFWWdQk8jl6Wmkl+r4hoY8zAPBgNVHRMB\nAf8EBTADAQH/MA0GCSqGSIb3DQEBCwUAA4ICAQBPv0q2OjExx4RypECI4C0LQtLo\njBrWitz7tIBN+pg5EJmSMfZqHypTvErX8ACEuWeV1pLmBHTrW/Y5OzVzslwjMGj0\nnzZaGj6+nQA+xP1rqD1uFIz8JLN9gkUBmzoitBqv1M06YKWKDMeY8FEqPoA4smQg\nsBCOw6G5jGLpNwOFF7mrWkGWL6GAiHno/XiDHQgOG+e8sflQu9VmZhJk6+E1Pbyw\neKtdWNxrr82KY32U+D8z2Q4x8EUhft4BEVbidN+l4mFaK9Dd7SXCYPeG8FL9ejcj\ncORGJ447d/vMlaHF4hCpO9VajkEXErPDaxeXk3YyUf55ngErG2j0q7JmkKHZfDNW\nxz4oUwq51FF1/zAlx25RNjfw+X01tToDQFORyZONTmtskBKpTQKTWTPBqV35dM1A\nycEwXRPUYDNkx8C5qBuIjo0m3Tg4ynczhBS24L2DSvXARdc53vmyQxH/dFD+3KTz\nvV+kVccGjzvbRCPnIuBMrKC1dISp4AH7V/aWtrYStlR9Dczyf35Dw9kBIBSuBGXF\nk0Y1sz2H4Y8bzPkQJYniQlMSNAE2u/IlaGDmNjU/Jz1HPT4HQw8yOCV2vPXsFTJa\nO/RBnXwv2OlD8ZovIe9Jj3wHjOiiC2F7jOUkG0AdezBL0OoI3aeeOuJtwgWe8xId\nmxkGBfwQH6Ut2F8VYQ==\n-----END CERTIFICATE-----\n"}';
	s_RootCA						: STRING(1283):= '-----BEGIN CERTIFICATE-----\nMIIDdzCCAl+gAwIBAgIUL1oQITunxPxaR4r6HQuPcRZeIUowDQYJKoZIhvcNAQEL\nBQAwSjEmMCQGA1UEAwwdVkVTIFNlbGYtc2lnbmVkIDE5Mi4xNjguMS4xMjYxCzAJ\nBgNVBAYTAk5MMRMwEQYDVQQHDApPdmVyaWpzc2VsMCAXDTI0MDMwNzE1MjU1MVoY\nDzIxMjEwODI2MTUyNTUxWjBKMSYwJAYDVQQDDB1WRVMgU2VsZi1zaWduZWQgMTky\nLjE2OC4xLjEyNjELMAkGA1UEBhMCTkwxEzARBgNVBAcMCk92ZXJpanNzZWwwggEi\nMA0GCSqGSIb3DQEBAQUAA4IBDwAwggEKAoIBAQC2HgB7KTx120GMtx+8fxY2VVm4\nXCz0WoIMgKeIbT7AHLH9FL6bEWiSCYdVWmLdSP53I32Amz93sjF6JRzxKVMM2OG5\n4ZkAKvejgePGWLRBL/kqf+0G3saga3lSCkmdJ9K+MRAGkE4WxcpnRZRQFZ46+7Fy\nfqfL+OWwazcNeTJp72l4D0BcPEJbgEuOIyOguUzSGitiK9nxMaq1rtIQ5Io/hg/J\nLfyjZ/Zha1V1qGco93410KyCSDpIF9L422by3mUOhn0AOMmfbMAk9XZmnGnbn7Pq\nIXtHEypEb7bcgAk7NehZHa+6bOyySEaxHcD888muRa458M/mpUG26fr7GOL9AgMB\nAAGjUzBRMB0GA1UdDgQWBBQut15Nm/Gnk4UsaVVK5LWEQWmilTAfBgNVHSMEGDAW\ngBQut15Nm/Gnk4UsaVVK5LWEQWmilTAPBgNVHRMBAf8EBTADAQH/MA0GCSqGSIb3\nDQEBCwUAA4IBAQCEc0xguZVreDCk1rFUJHSZqq3su8EbBhCTaCGrXLi2+ky7QnDm\nibHD29L9vyBPf/4kVY8dYOT0MwNb5qtfESyr7NMD/BTcnd7/zprGL7agWXbAO1xH\njw41vQW6dhd+GbUh9ftzHFrOiOnYKeUnISauyWD6yH8kFDjdaByU8r/lSJ23SXWE\nrDK8TSgKPRYYh4kH3snUPlscwivjZj9I8MiSx2GpqqogTrwNjoM/pVj+z2ENrUGR\nj0eWEJ2UiDxXtKhAQYOLyT7Nvmscb68CBVZPTv3sq+BvAkGPAQE8G7I38Nh+vEJ5\nVlFbMEjDO3FnkDx20dg53936N5w0x+Res2R4\n-----END CERTIFICATE-----\n';

	r_trigConnected					: R_TRIG;
	
	i_OnChangeValuesIndex			: INT;
END_VAR

VAR_IN_OUT CONSTANT
	{ attribute 'TcHmiSymbol.Hide' }
	monitor							: ST_System_Monitor;
END_VAR

VAR_IN_OUT 
	aData							: ARRAY [1..2000] OF ST_IoTDataHMI;
	controlvars						: ST_ExtController_get;
	st_params						: ST_IOT_params;
END_VAR

VAR_INPUT
	updateTrigger					: BOOL;
END_VAR

VAR
	updateList						: R_TRIG;
END_VAR

VAR_OUTPUT
	e_state							: eConnectionState;
END_VAR

VAR
	sJsonDocX8			:	STRING(2000);
	

	FastMessageState 		: ST_IOT_SentStateLog;
	SlowMessageState 		: ST_IOT_SentStateLog;
	DailyMessageState 		: ST_IOT_SentStateLog;
	OnchangeMessageState 	: ST_IOT_SentStateLog;
	aCheckSumLast			: ARRAY [1..2000] OF WORD;
END_VAR

// This script:
//   - Initializes an encrypted MQTT connection with openremote in the local network using the auto-provisioning method.
//   - Publishes data from the variables specified in the method "IotMapping", at different rates: Fast, Slow or OnChange (if ST_RW.WriteToNuc:=TRUE).
//   - Subcribes on topics as specified in the method "IotMapping" and pushes the received values back to the variable (if ST_RW.ReadFromNuc:=TRUE).
timer1(START:=TRUE,RESET:=TRUE);
rtrig_shutdownRequested(clk := w_shutdown = 1); //trigger instant message upon shutdown request
// -----( 0 )---------------------------  Prepare ------------------------------------------------------------------------------
// Clear previous received message
sMessage:=sMessageEmpty;

//Activate Timers
fbSendFastMessageTimer(IN:= NOT fbSendFastMessageTimer.Q, PT:= TO_TIME(st_params.r_UpdateTimeFast * 1000));
fbSendSlowMessageTimer(IN:= NOT fbSendSlowMessageTimer.Q, PT:= TO_TIME(st_params.r_UpdateTimeSlow * 1000));
fbDailyTimer(IN:= NOT fbDailyTimer.Q,);
fbConnectionTimer(IN:= NOT fbConnectionTimer.Q);

//-----( 1 )------------------- Initiate MQTT Connection using auto-provisioning------------------------------------------------
//------------------------------------------------------------------------------------------------------------------------------

IF (NOT fbMqttclient.bConnected AND fbConnectionTimer.Q) OR fbDailyTimer.Q THEN
	e_state := eConnectionState.disconnected;
	//Reset connection
	fbMqttClient.Execute(FALSE);
	//Configure
	IF bSetParameter THEN
		bSetParameter := FALSE;
		fbMqttClient.sHostName							:= '10.4.0.41';
		fbMqttClient.nHostPort							:= 8883;
		fbMqttClient.sTopicPrefix						:= '';
		fbMqttClient.sClientId							:= 'plc';
		fbMqttClient.sUserName							:= '';
		fbMqttClient.sUserPassword						:= '';
		fbMqttClient.stTLS.bNoServerCertCheck			:= TRUE;
		fbMqttClient.stTLS.sCA							:= 'c:\PLCUtility\rootCA.pem'; 
		fbMqttClient.nKeepAlive							:= 60;
		fbMqttClient.ipMessageQueue						:= fbMessageQueue;
	END_IF
	//Set and check, get error code
	fbMqttClient.Execute(bConnect);
	IF fbMqttClient.bError THEN
		hrErrorOccurred := fbMqttClient.hrErrorCode;
	END_IF	
    //Clear the Subscribe message structures
	stAutoProvisioning:=stAutoProvClear;

ELSE
	//Reset parameter set for next time connecting
	bSetParameter := TRUE;
END_IF

//Trigger connected state on rising edge
r_trigConnected(CLK:= fbMqttclient.bConnected);
IF r_trigConnected.Q THEN
	e_state := eConnectionState.connected;
END_IF

ConnectionState:= fbMQTTClient.eConnectionState;

//Auto Provisioning Pub/Sub		
IF	e_state < eConnectionState.authorized AND fbConnectionTimer.Q THEN
	//Subscribe on auto-provisioning channel
	IF NOT bSubscribedAutoProv THEN
		bSubscribedAutoProv:= fbMqttClient.Subscribe(sTopic:=autoProvSub,eQoS:=TcIotMqttQos.AtMostOnceDelivery);
	END_IF
	//Publish auto-provisioning request
	fbMqttClient.Publish(sTopic:=autoProvPub,
	pPayload := ADR(s_AutoProvMsg),
	nPayloadSize := LEN2(ADR(s_AutoProvMsg)),
	eQoS := TcIotMqttQos.AtMostOnceDelivery,
	bRetain:= FALSE,
	bQueue := FALSE);
	
	//Reset Asset Subscribtion Initialization
	bSubscribed:= FALSE;
	//Initiate on daily messages to be send one time after connect.
	DailyMessageState.bUpdate := TRUE;
	bInitiateFirstTimeSend := TRUE;

END_IF

//Start new Execute (else you won't receive messages...)
fbMqttClient.Execute(bConnect);

//Check for incomming messages
IF fbMessageQueue.nQueuedMessages > 0 THEN
	 IF fbMessageQueue.Dequeue(fbMessage:=fbMessage) THEN
		fbMessage.GetTopic(pTopic:=ADR(receivingTopic), nTopicSize:=SIZEOF(receivingTopic) );
		//Process autoprovisioning topic message
		IF receivingTopic = autoProvSub THEN
			fbMessage.GetPayload(pPayload:=ADR(sMessage), nPayloadSize:=SIZEOF(sMessage), bSetNullTermination:=FALSE );
			
			IF find(sMessage, 'success') <> 0 THEN
				e_state := eConnectionState.authorized;
			ELSIF find(sMessage, 'error') <> 0 THEN
				e_state := eConnectionState.authorization_declined;
			END_IF
//--------------------------------------END OF AUTO PROVISIONING---------------------------------------------------------
		ELSE
			// Process asset messages
			bIncommingMsg:=TRUE;
			fbMessage.GetPayload(pPayload:=ADR(sMessage), nPayloadSize:=SIZEOF(sMessage), bSetNullTermination:=FALSE);
			// OpenRemote sends attributevalue in extra quotes if it is a string, remove extra quotes (now double pressent)
			IF LEFT(sMessage,1)= '"' AND RIGHT(sMessage,1)= '"' THEN
			    sMessage:=DELETE(sMessage,1,1);
			    sMessage:=DELETE(sMessage,1,LEN(sMessage));
			END_IF
		END_IF
	END_IF
END_IF

//--------(  2  )----------Process Incomming Messages--------------------------------------------------------------------
//-----------------------------------------------------------------------------------------------------------------------

//Subscribe to Topics
iSizeTotal := MIN(TO_INT(eDataMappingVarNames.last), iSizeMax);
IF NOT bSubscribed AND e_state = eConnectionState.authorized THEN
		FOR i:= 1 TO iSizeTotal BY 1 DO
			IF NOT aData[i].b_IOTWriteAllowed THEN
				CONTINUE; // Jump to the next loop.
			END_IF
			//----Get variable mapping properties corresponding to index
			st_IotProps:= IotMappingV2(i);
			
			//----Check if topic is marked for subscribtion
			IF st_IotProps.st_RW.ReadFromNUC THEN
				sSubscribtion:=concat(concat(sSubPreFix,st_IotProps.sName),sAssetID);
				fbMqttClient.Subscribe(sTopic:=sSubscribtion,eQoS:=TcIotMqttQos.AtMostOnceDelivery);
			END_IF			
		END_FOR
	bSubscribed:=TRUE;
END_IF

//Process Received Messages
IF e_state = eConnectionState.authorized AND bIncommingMsg THEN
	FOR i:= 1 TO iSizeTotal BY 1 DO
		//Check if data write is enabled:
		IF NOT aData[i].b_IOTWriteAllowed THEN
			CONTINUE; // Jump to the next loop.
		END_IF
		
		st_IotProps:= IotMappingV2(i);
		//----Make the topic in format as is received for comparison
		sSubChecker:= concat(concat(sSubPrefix,st_IotProps.sName),sAssetID);
		//Check if the received message corresponds to the current index 
		IF receivingTopic = sSubChecker AND st_IotProps.st_RW.ReadFromNUC THEN
			//Put payload into variable
			IotWriteBackToVar(sMessage,st_IotProps.pAdress,st_IotProps.ClassType);
			//Disable processing again.
			bIncommingMsg:=FALSE;
		END_IF
	END_FOR
END_IF

//-----  (  3  ) ----------Publish Messages based on IotMapping and Fast, Slow or OnChange timers------------------------
//-----------------------------------------------------------------------------------------------------------------------

updatelist(CLK := UpdateTrigger);
IF updateList.Q THEN
	SlowMessageState.LastIndex := 0;
	FastMessageState.LastIndex := 0;
	DailyMessageState.LastIndex := 0;
	OnchangeMessageState.LastIndex := 0;
	FOR i := 1 TO iSizeTotal DO
		//---- Determine last index of fast and slow variables
		IF aData[i].LogInterval = eUpdate.Fast AND aData[i].LogType <> eLogType.none THEN
			FastMessageState.LastIndex := i;
		END_IF
		IF aData[i].LogInterval = eUpdate.Slow AND aData[i].LogType <> eLogType.none THEN
			SlowMessageState.LastIndex := i;
		END_IF
		IF aData[i].LogInterval = eUpdate.Daily AND aData[i].LogType <> eLogType.none THEN
			DailyMessageState.LastIndex := i;
		END_IF
		IF aData[i].LogInterval = eUpdate.Onchange AND aData[i].LogType <> eLogType.none THEN
			OnchangeMessageState.LastIndex := i;
		END_IF
	END_FOR
END_IF

b_UpdateActive := rtrig_shutdownRequested.q;

IF fbSendFastMessageTimer.Q THEN
	FastMessageState.bUpdate := TRUE;
END_IF
IF fbSendSlowMessageTimer.Q THEN
	SlowMessageState.bUpdate := TRUE;
END_IF
IF fbSendFastMessageTimer.Q  OR DailyMessageState.bUpdate OR rtrig_shutdownRequested.q THEN
	OnchangeMessageState.bUpdate := TRUE;
END_IF

IF controlvars.LoggingBudgetOK THEN
	PublishVarsV2(Authorized := e_state = eConnectionState.authorized, interval := eUpdate.Fast, state := FastMessageState);
	PublishVarsV2(Authorized := e_state = eConnectionState.authorized, interval := eUpdate.Slow, state := SlowMessageState);
	PublishVarsV2(Authorized := e_state = eConnectionState.authorized, interval := eUpdate.Daily, state := DailyMessageState);
	PublishVarsV2(Authorized := e_state = eConnectionState.authorized, interval := eUpdate.onchange, state := OnchangeMessageState);
end_if
PublishVarsV1();

timer1(START:=FALSE);

controlvars.e_ConnectionState := e_state;

METHOD PUBLIC FillBatteryDatalog : BOOL
VAR_INPUT
	s_MBMUData	:	STRING(255);
	s_SBMUData	:	ARRAY[0..3] OF STRING (255);
	s_EMSData	:	STRING(255);
END_VAR

VAR
	fbJson      	: FB_JsonSaxWriter;
END_VAR
fbJson.StartObject();
fbJson.AddKeyString('MBMU',s_MBMUData);
fbJson.AddKeyString('SBMU1',s_SBMUData[0]);
fbJson.AddKeyString('SBMU2',s_SBMUData[1]);
fbJson.AddKeyString('SBMU3',s_SBMUData[2]);
fbJson.AddKeyString('SBMU4',s_SBMUData[3]);
fbJson.AddKeyString('EMS',s_EMSData);
fbJson.EndObject();
fbJson.CopyDocument(pDoc := sJsonDocX8, nDoc := SIZEOF(sJsonDocX8));
END_METHOD

METHOD IoTExtractType : ST_VarBuffer
VAR_INPUT
	sVariableName	: ANY;
	precision		: INT := 0; 
	threshold		: REAL := 0;
END_VAR

VAR
	bNumber		: BOOL;
	
	tempReal	: REAL;
	tempLreal	: LREAL;
	tempDword	: DWORD;
	tempWord	: WORD;
	tempSINT	: SINT;
	tempint		: INT;
	tempUint	: UINT;
	tempusint	: USINT;
	//pTosValue	: PVOID := ADR(sValue);
END_VAR
CASE UDINT_TO_INT(sVariableName.TypeClass) OF
    IBaseLibrary.TypeClass.TYPE_BOOL :
		IF PBOOL_TO_BOOL(sVariableName.pValue) THEN
			IotExtractType.sValue := 'true';
		ELSIF NOT PBOOL_TO_BOOL(sVariableName.pValue) THEN
			IotExtractType.sValue := 'false';
		END_IF
		bNumber:= TRUE;
    IBaseLibrary.TypeClass.TYPE_ENUM :
		IotExtractType.sValue	:= TO_STRING(PINT_TO_INT(sVariableName.pValue));
		bNumber:= FALSE;
    IBaseLibrary.TypeClass.TYPE_LREAL :
		tempLreal := PLREAL_TO_LREAL(sVariableName.pValue);
		IF ABS(tempLreal) < threshold THEN tempLreal := 0; END_IF
		IotExtractType.sValue	:= TO_STRING(LREAL_TO_FMTSTR(tempLreal, precision, TRUE));
		bNumber:= TRUE;
    IBaseLibrary.TypeClass.TYPE_WORD :
		tempword := PWORD_TO_WORD(sVariableName.pValue);
		IF tempword < threshold THEN tempword := 0; END_IF
		IotExtractType.sValue	:= TO_STRING(tempword);
		bNumber:= TRUE;
    IBaseLibrary.TypeClass.TYPE_DWORD :
		tempDword := PDWORD_TO_DWORD(sVariableName.pValue);
		IF tempdword < threshold THEN tempdword := 0; END_IF
		IotExtractType.sValue	:= TO_STRING(tempdword);
		bNumber:= TRUE;
    IBaseLibrary.TypeClass.TYPE_SINT :
		tempsint := PSINT_TO_SINT(sVariableName.pValue);
		IF ABS(tempsint) < threshold THEN tempsint := 0; END_IF
		IotExtractType.sValue	:= TO_STRING(tempsint);
		bNumber:= TRUE;
    IBaseLibrary.TypeClass.TYPE_INT :
		tempint := PINT_TO_INT(sVariableName.pValue);
		IF ABS(tempint) < threshold THEN tempint := 0; END_IF
		IotExtractType.sValue	:= TO_STRING(tempint);
		bNumber:= TRUE;	
	IBaseLibrary.TypeClass.TYPE_UINT :
		tempuint := PUINT_TO_UINT(sVariableName.pValue);
		IF tempuint < threshold THEN tempuint := 0; END_IF
		IotExtractType.sValue	:= TO_STRING(tempuint);
		bNumber:= TRUE;	
    IBaseLibrary.TypeClass.TYPE_REAL :
		tempreal := PREAL_TO_REAL(sVariableName.pValue);
		IF ABS(tempreal) < threshold THEN tempreal := 0; END_IF
		IotExtractType.sValue	:= TO_STRING(LREAL_TO_FMTSTR(tempreal, precision, TRUE));
		bNumber:= TRUE;
	IBaseLibrary.TypeClass.TYPE_STRING :
		//Pas op gevaarlijke functie, doet rechtstreeks geheugen adres manipulatie!
		memcpy(ADR(IotExtractType.sValue),sVariableName.pValue,sVariablename.diSize);
		bNumber:= FALSE;
	IBaseLibrary.TypeClass.TYPE_USINT :
		tempusint := PUSINT_TO_USINT(sVariableName.pValue);
		IF tempusint < threshold THEN tempusint := 0; END_IF
		IotExtractType.sValue	:= TO_STRING(tempusint);
		bNumber:= TRUE;
ELSE
	IotExtractType.sValue:='UNKNOWN_DATA_TYPE';
		
END_CASE

IoTExtractType.pAdress	:= sVariableName.pValue;
IotExtractType.diSize := sVariableName.diSize;
IotExtractType.ClassType:= sVariableName.TypeClass;
IotExtractType.bNumber  := bNumber;
END_METHOD

METHOD IotMapping : ST_IotProps
VAR_INPUT
	index : INT;
END_VAR

VAR
	pAdress 		: PVOID;
	st_Variable		: ST_VarBuffer;
	bJson			: BOOL;
	tempString		: STRING;
	tempReal		: REAL;
	fbJson      	: FB_JsonSaxWriter;
	sJsonDocX12     : STRING(255);
	sJsonDocX11     : STRING(255);
	
	jsonKey			: STRING;
	i				: INT; // for loop index
	
END_VAR

